        OnMouseDown: execute { SR_MulticarrierModule.udiSingleCarrierNr := 131; }
    Button (68,712 25x25), "132", colour toggle: SR_MulticarrierModule.aifVisFeedback[132].ifFeedbackConfiguration.xApplicationLoggerEntriesActive, invisible if: SR_MulticarrierModule.ifMulticarrier.ifFeedback.ifFeedbackConfiguration.udiNumberOfCarriers < 132
        toggle SR_MulticarrierModule.xSetSingleAplMsg
        OnMouseDown: execute { SR_MulticarrierModule.udiSingleCarrierNr := 132; }
    Button (108,712 25x25), "133", colour toggle: SR_MulticarrierModule.aifVisFeedback[133].ifFeedbackConfiguration.xApplicationLoggerEntriesActive, invisible if: SR_MulticarrierModule.ifMulticarrier.ifFeedback.ifFeedbackConfiguration.udiNumberOfCarriers < 133
        toggle SR_MulticarrierModule.xSetSingleAplMsg
        OnMouseDown: execute { SR_MulticarrierModule.udiSingleCarrierNr := 133; }
    Button (148,712 25x25), "134", colour toggle: SR_MulticarrierModule.aifVisFeedback[134].ifFeedbackConfiguration.xApplicationLoggerEntriesActive, invisible if: SR_MulticarrierModule.ifMulticarrier.ifFeedback.ifFeedbackConfiguration.udiNumberOfCarriers < 134
        toggle SR_MulticarrierModule.xSetSingleAplMsg
        OnMouseDown: execute { SR_MulticarrierModule.udiSingleCarrierNr := 134; }
    Button (188,712 25x25), "135", colour toggle: SR_MulticarrierModule.aifVisFeedback[135].ifFeedbackConfiguration.xApplicationLoggerEntriesActive, invisible if: SR_MulticarrierModule.ifMulticarrier.ifFeedback.ifFeedbackConfiguration.udiNumberOfCarriers < 135
        toggle SR_MulticarrierModule.xSetSingleAplMsg
        OnMouseDown: execute { SR_MulticarrierModule.udiSingleCarrierNr := 135; }
    Button (228,712 25x25), "136", colour toggle: SR_MulticarrierModule.aifVisFeedback[136].ifFeedbackConfiguration.xApplicationLoggerEntriesActive, invisible if: SR_MulticarrierModule.ifMulticarrier.ifFeedback.ifFeedbackConfiguration.udiNumberOfCarriers < 136
        toggle SR_MulticarrierModule.xSetSingleAplMsg
        OnMouseDown: execute { SR_MulticarrierModule.udiSingleCarrierNr := 136; }
    Button (268,712 25x25), "137", colour toggle: SR_MulticarrierModule.aifVisFeedback[137].ifFeedbackConfiguration.xApplicationLoggerEntriesActive, invisible if: SR_MulticarrierModule.ifMulticarrier.ifFeedback.ifFeedbackConfiguration.udiNumberOfCarriers < 137
        toggle SR_MulticarrierModule.xSetSingleAplMsg
        OnMouseDown: execute { SR_MulticarrierModule.udiSingleCarrierNr := 137; }
    Button (308,712 25x25), "138", colour toggle: SR_MulticarrierModule.aifVisFeedback[138].ifFeedbackConfiguration.xApplicationLoggerEntriesActive, invisible if: SR_MulticarrierModule.ifMulticarrier.ifFeedback.ifFeedbackConfiguration.udiNumberOfCarriers < 138
        toggle SR_MulticarrierModule.xSetSingleAplMsg
        OnMouseDown: execute { SR_MulticarrierModule.udiSingleCarrierNr := 138; }
    Button (348,712 25x25), "139", colour toggle: SR_MulticarrierModule.aifVisFeedback[139].ifFeedbackConfiguration.xApplicationLoggerEntriesActive, invisible if: SR_MulticarrierModule.ifMulticarrier.ifFeedback.ifFeedbackConfiguration.udiNumberOfCarriers < 139
        toggle SR_MulticarrierModule.xSetSingleAplMsg
        OnMouseDown: execute { SR_MulticarrierModule.udiSingleCarrierNr := 139; }
    Button (387,712 25x25), "140", colour toggle: SR_MulticarrierModule.aifVisFeedback[140].ifFeedbackConfiguration.xApplicationLoggerEntriesActive, invisible if: SR_MulticarrierModule.ifMulticarrier.ifFeedback.ifFeedbackConfiguration.udiNumberOfCarriers < 140
        toggle SR_MulticarrierModule.xSetSingleAplMsg
        OnMouseDown: execute { SR_MulticarrierModule.udiSingleCarrierNr := 140; }
    Button (27,752 25x25), "141", colour toggle: SR_MulticarrierModule.aifVisFeedback[141].ifFeedbackConfiguration.xApplicationLoggerEntriesActive, invisible if: SR_MulticarrierModule.ifMulticarrier.ifFeedback.ifFeedbackConfiguration.udiNumberOfCarriers < 141
        toggle SR_MulticarrierModule.xSetSingleAplMsg
        OnMouseDown: execute { SR_MulticarrierModule.udiSingleCarrierNr := 141; }
    Button (67,752 25x25), "142", colour toggle: SR_MulticarrierModule.aifVisFeedback[142].ifFeedbackConfiguration.xApplicationLoggerEntriesActive, invisible if: SR_MulticarrierModule.ifMulticarrier.ifFeedback.ifFeedbackConfiguration.udiNumberOfCarriers < 142
        toggle SR_MulticarrierModule.xSetSingleAplMsg
        OnMouseDown: execute { SR_MulticarrierModule.udiSingleCarrierNr := 142; }
    Button (107,752 25x25), "143", colour toggle: SR_MulticarrierModule.aifVisFeedback[143].ifFeedbackConfiguration.xApplicationLoggerEntriesActive, invisible if: SR_MulticarrierModule.ifMulticarrier.ifFeedback.ifFeedbackConfiguration.udiNumberOfCarriers < 143
        toggle SR_MulticarrierModule.xSetSingleAplMsg
        OnMouseDown: execute { SR_MulticarrierModule.udiSingleCarrierNr := 143; }
    Button (147,752 25x25), "144", colour toggle: SR_MulticarrierModule.aifVisFeedback[144].ifFeedbackConfiguration.xApplicationLoggerEntriesActive, invisible if: SR_MulticarrierModule.ifMulticarrier.ifFeedback.ifFeedbackConfiguration.udiNumberOfCarriers < 144
        toggle SR_MulticarrierModule.xSetSingleAplMsg
        OnMouseDown: execute { SR_MulticarrierModule.udiSingleCarrierNr := 144; }
    Button (187,752 25x25), "145", colour toggle: SR_MulticarrierModule.aifVisFeedback[145].ifFeedbackConfiguration.xApplicationLoggerEntriesActive, invisible if: SR_MulticarrierModule.ifMulticarrier.ifFeedback.ifFeedbackConfiguration.udiNumberOfCarriers < 145
        toggle SR_MulticarrierModule.xSetSingleAplMsg
        OnMouseDown: execute { SR_MulticarrierModule.udiSingleCarrierNr := 145; }
    Button (227,752 25x25), "146", colour toggle: SR_MulticarrierModule.aifVisFeedback[146].ifFeedbackConfiguration.xApplicationLoggerEntriesActive, invisible if: SR_MulticarrierModule.ifMulticarrier.ifFeedback.ifFeedbackConfiguration.udiNumberOfCarriers < 146
        toggle SR_MulticarrierModule.xSetSingleAplMsg
        OnMouseDown: execute { SR_MulticarrierModule.udiSingleCarrierNr := 146; }
    Button (267,752 25x25), "147", colour toggle: SR_MulticarrierModule.aifVisFeedback[147].ifFeedbackConfiguration.xApplicationLoggerEntriesActive, invisible if: SR_MulticarrierModule.ifMulticarrier.ifFeedback.ifFeedbackConfiguration.udiNumberOfCarriers < 147
        toggle SR_MulticarrierModule.xSetSingleAplMsg
        OnMouseDown: execute { SR_MulticarrierModule.udiSingleCarrierNr := 147; }
    Button (307,752 25x25), "148", colour toggle: SR_MulticarrierModule.aifVisFeedback[148].ifFeedbackConfiguration.xApplicationLoggerEntriesActive, invisible if: SR_MulticarrierModule.ifMulticarrier.ifFeedback.ifFeedbackConfiguration.udiNumberOfCarriers < 148
        toggle SR_MulticarrierModule.xSetSingleAplMsg
        OnMouseDown: execute { SR_MulticarrierModule.udiSingleCarrierNr := 148; }
    Button (347,752 25x25), "149", colour toggle: SR_MulticarrierModule.aifVisFeedback[149].ifFeedbackConfiguration.xApplicationLoggerEntriesActive, invisible if: SR_MulticarrierModule.ifMulticarrier.ifFeedback.ifFeedbackConfiguration.udiNumberOfCarriers < 149
        toggle SR_MulticarrierModule.xSetSingleAplMsg
        OnMouseDown: execute { SR_MulticarrierModule.udiSingleCarrierNr := 149; }
    Button (388,752 25x25), "150", colour toggle: SR_MulticarrierModule.aifVisFeedback[150].ifFeedbackConfiguration.xApplicationLoggerEntriesActive, invisible if: SR_MulticarrierModule.ifMulticarrier.ifFeedback.ifFeedbackConfiguration.udiNumberOfCarriers < 150
        toggle SR_MulticarrierModule.xSetSingleAplMsg
        OnMouseDown: execute { SR_MulticarrierModule.udiSingleCarrierNr := 150; }
    Button (188,672 25x25), "125", colour toggle: SR_MulticarrierModule.aifVisFeedback[125].ifFeedbackConfiguration.xApplicationLoggerEntriesActive, invisible if: SR_MulticarrierModule.ifMulticarrier.ifFeedback.ifFeedbackConfiguration.udiNumberOfCarriers < 125
        toggle SR_MulticarrierModule.xSetSingleAplMsg
        OnMouseDown: execute { SR_MulticarrierModule.udiSingleCarrierNr := 125; }
    Button (228,672 25x25), "126", colour toggle: SR_MulticarrierModule.aifVisFeedback[126].ifFeedbackConfiguration.xApplicationLoggerEntriesActive, invisible if: SR_MulticarrierModule.ifMulticarrier.ifFeedback.ifFeedbackConfiguration.udiNumberOfCarriers < 126
        toggle SR_MulticarrierModule.xSetSingleAplMsg
        OnMouseDown: execute { SR_MulticarrierModule.udiSingleCarrierNr := 126; }
    Button (268,672 25x25), "127", colour toggle: SR_MulticarrierModule.aifVisFeedback[127].ifFeedbackConfiguration.xApplicationLoggerEntriesActive, invisible if: SR_MulticarrierModule.ifMulticarrier.ifFeedback.ifFeedbackConfiguration.udiNumberOfCarriers < 127
        toggle SR_MulticarrierModule.xSetSingleAplMsg
        OnMouseDown: execute { SR_MulticarrierModule.udiSingleCarrierNr := 127; }
    Button (308,672 25x25), "128", colour toggle: SR_MulticarrierModule.aifVisFeedback[128].ifFeedbackConfiguration.xApplicationLoggerEntriesActive, invisible if: SR_MulticarrierModule.ifMulticarrier.ifFeedback.ifFeedbackConfiguration.udiNumberOfCarriers < 128
        toggle SR_MulticarrierModule.xSetSingleAplMsg
        OnMouseDown: execute { SR_MulticarrierModule.udiSingleCarrierNr := 128; }
    Button (348,672 25x25), "129", colour toggle: SR_MulticarrierModule.aifVisFeedback[129].ifFeedbackConfiguration.xApplicationLoggerEntriesActive, invisible if: SR_MulticarrierModule.ifMulticarrier.ifFeedback.ifFeedbackConfiguration.udiNumberOfCarriers < 129
        toggle SR_MulticarrierModule.xSetSingleAplMsg
        OnMouseDown: execute { SR_MulticarrierModule.udiSingleCarrierNr := 129; }
    Rectangle (339,110 100x20), "End: %0.0f", text variable: SR_MulticarrierModule.lrAplEndTrackPos
        OnMouseClick: write the text variable via Default, min 0, max SR_MulticarrierModule.fbMulticarrier.ifFeedback.ifFeedbackConfiguration.lrTrackLength
    Button (339,49 100x40), "Set entries by Position", colour toggle: SR_MultiCarriermodule.xAplMsgStartPosAndEndPos
        toggle SR_MultiCarriermodule.xAplMsgStartPosAndEndPos
    Rectangle (339,90 100x20), "Start: %0.0f", text variable: SR_MulticarrierModule.lrAplStartTrackPos
        OnMouseClick: write the text variable via Default, min 0, max SR_MulticarrierModule.fbMulticarrier.ifFeedback.ifFeedbackConfiguration.lrTrackLength
END_VISUALIZATION

// LMC_PacDrive/Application/TemplateFullProgrammingFramework/Visualization/Multicarrier/Vis_Error
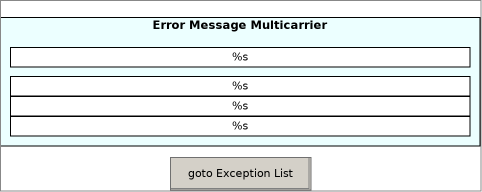
VISUALIZATION Vis_Error  // 482x192
    Rectangle (0,17 480x129), "Error Message Multicarrier"
    Rectangle (10,47 460x20), "%s", text variable: SR_MultiCarrierModule.stException.sDiagExt
    Rectangle (10,76 460x20), "%s", text variable: SR_MultiCarrierModule.sResultMsg1
    Rectangle (10,96 460x20), "%s", text variable: SR_MultiCarrierModule.sResultMsg2
    Button (170,157 141x33), "goto Exception List"
        OnMouseClick:  Assign=VIS_ExceptionList, Type=Assignment
    Rectangle (10,116 460x20), "%s", text variable: SR_MultiCarrierModule.sResultMsg3
END_VISUALIZATION

// LMC_PacDrive/Application/TemplateFullProgrammingFramework/Visualization/Multicarrier/Vis_Jogging
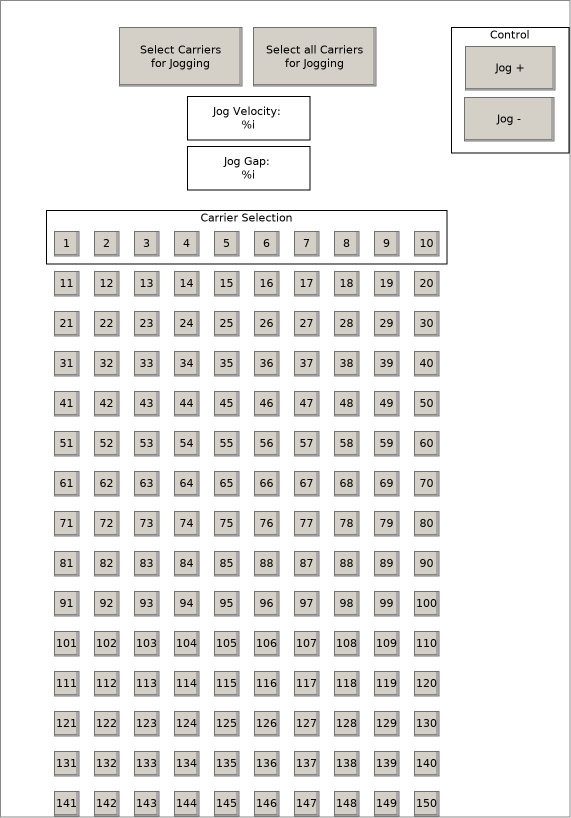
VISUALIZATION Vis_Jogging  // 571x818
    Rectangle (451,27 118x126), "Control", input disabled if: NOT SR_MainMachine.xActManual
    Button (465,46 90x44), "Jog +", colour toggle: SR_MulticarrierModule.xJogForw, input disabled if: NOT SR_MainMachine.xActManual
        tap SR_MulticarrierModule.xJogForw
    Button (464,97 90x44), "Jog -", colour toggle: SR_MulticarrierModule.xJogBack, input disabled if: NOT SR_MainMachine.xActManual
        tap SR_MulticarrierModule.xJogBack p3779583253=TRUE
    Button (119,27 123x59), "Select Carriers for Jogging", colour toggle: SR_MulticarrierModule.xJogSingleCarrier, input disabled if: NOT SR_MainMachine.xActManual
        tap SR_MultiCarriermodule.xSetJogSingleCarrier
    Button (253,27 123x59), "Select all Carriers for Jogging", colour toggle: SR_MulticarrierModule.xJogAllCarrier, input disabled if: NOT SR_MainMachine.xActManual
        tap SR_MulticarrierModule.xSetJogAllCarrier
    Rectangle (187,96 123x44), "Jog Velocity: %i", tooltip "Acc = Velocity Dec = Velocity x 10 Jerk = Velocity x 100", text variable: SR_MulticarrierModule.lrJogVelocity, input disabled if: NOT SR_MainMachine.xActManual
        OnMouseClick: write the text variable via Default, min 0
    Rectangle (187,146 123x44), "Jog Gap: %i", tooltip "Jog possible when Actual Gap >= Jog Gap (Decelerate moving Carrier when Actual Gap < Jog Gap)", text variable: SR_MulticarrierModule.lrJogMinDistanceBetweenCarrier, invisible if: SR_MulticarrierModule.xJogAllCarrier, input disabled if: NOT SR_MainMachine.xActManual
        OnMouseClick: write the text variable via Default, min 0
    Rectangle (46,210 401x54), "Carrier Selection"
        p1126004900: SR_MultiCarriermodule.udiDeltaBottomY
    Button (54,231 25x25), "1", colour toggle: SR_MultiCarrierModule.aifVisFeedback[1].ifFeedbackJogging.xJogActivated, invisible if: SR_MulticarrierModule.ifMulticarrier.ifFeedback.ifFeedbackConfiguration.udiNumberOfCarriers < 1, input disabled if: NOT SR_MainMachine.xActManual
        toggle SR_MultiCarriermodule.xSetCarrierForJoggingFromVis
        OnMouseClick: execute { SR_MultiCarrierModule.udiJoggingCarrierNr := 1; }
    Button (94,231 25x25), "2", colour toggle: SR_MultiCarrierModule.aifVisFeedback[2].ifFeedbackJogging.xJogActivated, invisible if: SR_MulticarrierModule.ifMulticarrier.ifFeedback.ifFeedbackConfiguration.udiNumberOfCarriers < 2, input disabled if: NOT SR_MainMachine.xActManual
        toggle SR_MultiCarriermodule.xSetCarrierForJoggingFromVis
        OnMouseClick: execute { SR_MultiCarrierModule.udiJoggingCarrierNr := 2; }
    Button (134,231 25x25), "3", colour toggle: SR_MultiCarrierModule.aifVisFeedback[3].ifFeedbackJogging.xJogActivated, invisible if: SR_MulticarrierModule.ifMulticarrier.ifFeedback.ifFeedbackConfiguration.udiNumberOfCarriers < 3, input disabled if: NOT SR_MainMachine.xActManual
        toggle SR_MultiCarriermodule.xSetCarrierForJoggingFromVis
        OnMouseClick: execute { SR_MultiCarrierModule.udiJoggingCarrierNr := 3; }
    Button (174,231 25x25), "4", colour toggle: SR_MultiCarrierModule.aifVisFeedback[4].ifFeedbackJogging.xJogActivated, invisible if: SR_MulticarrierModule.ifMulticarrier.ifFeedback.ifFeedbackConfiguration.udiNumberOfCarriers < 4, input disabled if: NOT SR_MainMachine.xActManual
        toggle SR_MultiCarriermodule.xSetCarrierForJoggingFromVis
        OnMouseClick: execute { SR_MultiCarrierModule.udiJoggingCarrierNr := 4; }
    Button (214,231 25x25), "5", colour toggle: SR_MultiCarrierModule.aifVisFeedback[5].ifFeedbackJogging.xJogActivated, invisible if: SR_MulticarrierModule.ifMulticarrier.ifFeedback.ifFeedbackConfiguration.udiNumberOfCarriers < 5, input disabled if: NOT SR_MainMachine.xActManual
        toggle SR_MultiCarriermodule.xSetCarrierForJoggingFromVis
        OnMouseClick: execute { SR_MultiCarrierModule.udiJoggingCarrierNr := 5; }
    Button (254,231 25x25), "6", colour toggle: SR_MultiCarrierModule.aifVisFeedback[6].ifFeedbackJogging.xJogActivated, invisible if: SR_MulticarrierModule.ifMulticarrier.ifFeedback.ifFeedbackConfiguration.udiNumberOfCarriers < 6, input disabled if: NOT SR_MainMachine.xActManual
        toggle SR_MultiCarriermodule.xSetCarrierForJoggingFromVis
        OnMouseClick: execute { SR_MultiCarrierModule.udiJoggingCarrierNr := 6; }
    Button (294,231 25x25), "7", colour toggle: SR_MultiCarrierModule.aifVisFeedback[7].ifFeedbackJogging.xJogActivated, invisible if: SR_MulticarrierModule.ifMulticarrier.ifFeedback.ifFeedbackConfiguration.udiNumberOfCarriers < 7, input disabled if: NOT SR_MainMachine.xActManual
        toggle SR_MultiCarriermodule.xSetCarrierForJoggingFromVis
        OnMouseClick: execute { SR_MultiCarrierModule.udiJoggingCarrierNr := 7; }
    Button (334,231 25x25), "8", colour toggle: SR_MultiCarrierModule.aifVisFeedback[8].ifFeedbackJogging.xJogActivated, invisible if: SR_MulticarrierModule.ifMulticarrier.ifFeedback.ifFeedbackConfiguration.udiNumberOfCarriers < 8, input disabled if: NOT SR_MainMachine.xActManual
        toggle SR_MultiCarriermodule.xSetCarrierForJoggingFromVis
        OnMouseClick: execute { SR_MultiCarrierModule.udiJoggingCarrierNr := 8; }
    Button (374,231 25x25), "9", colour toggle: SR_MultiCarrierModule.aifVisFeedback[9].ifFeedbackJogging.xJogActivated, invisible if: SR_MulticarrierModule.ifMulticarrier.ifFeedback.ifFeedbackConfiguration.udiNumberOfCarriers < 9, input disabled if: NOT SR_MainMachine.xActManual
        toggle SR_MultiCarriermodule.xSetCarrierForJoggingFromVis
        OnMouseClick: execute { SR_MultiCarrierModule.udiJoggingCarrierNr := 9; }
    Button (414,231 25x25), "10", colour toggle: SR_MultiCarrierModule.aifVisFeedback[10].ifFeedbackJogging.xJogActivated, invisible if: SR_MulticarrierModule.ifMulticarrier.ifFeedback.ifFeedbackConfiguration.udiNumberOfCarriers < 10, input disabled if: NOT SR_MainMachine.xActManual
        toggle SR_MultiCarriermodule.xSetCarrierForJoggingFromVis
        OnMouseClick: execute { SR_MultiCarrierModule.udiJoggingCarrierNr := 10; }
    Button (414,271 25x25), "20", colour toggle: SR_MultiCarrierModule.aifVisFeedback[20].ifFeedbackJogging.xJogActivated, invisible if: SR_MulticarrierModule.ifMulticarrier.ifFeedback.ifFeedbackConfiguration.udiNumberOfCarriers < 20, input disabled if: NOT SR_MainMachine.xActManual
        toggle SR_MultiCarriermodule.xSetCarrierForJoggingFromVis
        OnMouseClick: execute { SR_MultiCarrierModule.udiJoggingCarrierNr := 20; }
    Button (414,311 25x25), "30", colour toggle: SR_MultiCarrierModule.aifVisFeedback[30].ifFeedbackJogging.xJogActivated, invisible if: SR_MulticarrierModule.ifMulticarrier.ifFeedback.ifFeedbackConfiguration.udiNumberOfCarriers < 30, input disabled if: NOT SR_MainMachine.xActManual
        toggle SR_MultiCarriermodule.xSetCarrierForJoggingFromVis
        OnMouseClick: execute { SR_MultiCarrierModule.udiJoggingCarrierNr := 30; }
    Button (414,351 25x25), "40", colour toggle: SR_MultiCarrierModule.aifVisFeedback[40].ifFeedbackJogging.xJogActivated, invisible if: SR_MulticarrierModule.ifMulticarrier.ifFeedback.ifFeedbackConfiguration.udiNumberOfCarriers < 40, input disabled if: NOT SR_MainMachine.xActManual
        toggle SR_MultiCarriermodule.xSetCarrierForJoggingFromVis
        OnMouseClick: execute { SR_MultiCarrierModule.udiJoggingCarrierNr := 40; }
    Button (414,391 25x25), "50", colour toggle: SR_MultiCarrierModule.aifVisFeedback[50].ifFeedbackJogging.xJogActivated, invisible if: SR_MulticarrierModule.ifMulticarrier.ifFeedback.ifFeedbackConfiguration.udiNumberOfCarriers < 50, input disabled if: NOT SR_MainMachine.xActManual
        toggle SR_MultiCarriermodule.xSetCarrierForJoggingFromVis
        OnMouseClick: execute { SR_MultiCarrierModule.udiJoggingCarrierNr := 50; }
    Button (414,431 25x25), "60", colour toggle: SR_MultiCarrierModule.aifVisFeedback[60].ifFeedbackJogging.xJogActivated, invisible if: SR_MulticarrierModule.ifMulticarrier.ifFeedback.ifFeedbackConfiguration.udiNumberOfCarriers < 60, input disabled if: NOT SR_MainMachine.xActManual
        toggle SR_MultiCarriermodule.xSetCarrierForJoggingFromVis
        OnMouseClick: execute { SR_MultiCarrierModule.udiJoggingCarrierNr := 60; }
    Button (54,471 25x25), "61", colour toggle: SR_MultiCarrierModule.aifVisFeedback[61].ifFeedbackJogging.xJogActivated, invisible if: SR_MulticarrierModule.ifMulticarrier.ifFeedback.ifFeedbackConfiguration.udiNumberOfCarriers < 61, input disabled if: NOT SR_MainMachine.xActManual
        toggle SR_MultiCarriermodule.xSetCarrierForJoggingFromVis
        OnMouseClick: execute { SR_MultiCarrierModule.udiJoggingCarrierNr := 61; }
    Button (94,471 25x25), "62", colour toggle: SR_MultiCarrierModule.aifVisFeedback[62].ifFeedbackJogging.xJogActivated, invisible if: SR_MulticarrierModule.ifMulticarrier.ifFeedback.ifFeedbackConfiguration.udiNumberOfCarriers < 62, input disabled if: NOT SR_MainMachine.xActManual
        toggle SR_MultiCarriermodule.xSetCarrierForJoggingFromVis
        OnMouseClick: execute { SR_MultiCarrierModule.udiJoggingCarrierNr := 62; }
    Button (134,471 25x25), "63", colour toggle: SR_MultiCarrierModule.aifVisFeedback[63].ifFeedbackJogging.xJogActivated, invisible if: SR_MulticarrierModule.ifMulticarrier.ifFeedback.ifFeedbackConfiguration.udiNumberOfCarriers < 63, input disabled if: NOT SR_MainMachine.xActManual
        toggle SR_MultiCarriermodule.xSetCarrierForJoggingFromVis
        OnMouseClick: execute { SR_MultiCarrierModule.udiJoggingCarrierNr := 63; }
    Button (174,471 25x25), "64", colour toggle: SR_MultiCarrierModule.aifVisFeedback[64].ifFeedbackJogging.xJogActivated, invisible if: SR_MulticarrierModule.ifMulticarrier.ifFeedback.ifFeedbackConfiguration.udiNumberOfCarriers < 64, input disabled if: NOT SR_MainMachine.xActManual
        toggle SR_MultiCarriermodule.xSetCarrierForJoggingFromVis
        OnMouseClick: execute { SR_MultiCarrierModule.udiJoggingCarrierNr := 64; }
    Button (214,471 25x25), "65", colour toggle: SR_MultiCarrierModule.aifVisFeedback[65].ifFeedbackJogging.xJogActivated, invisible if: SR_MulticarrierModule.ifMulticarrier.ifFeedback.ifFeedbackConfiguration.udiNumberOfCarriers < 65, input disabled if: NOT SR_MainMachine.xActManual
        toggle SR_MultiCarriermodule.xSetCarrierForJoggingFromVis
        OnMouseClick: execute { SR_MultiCarrierModule.udiJoggingCarrierNr := 65; }
    Button (254,471 25x25), "66", colour toggle: SR_MultiCarrierModule.aifVisFeedback[66].ifFeedbackJogging.xJogActivated, invisible if: SR_MulticarrierModule.ifMulticarrier.ifFeedback.ifFeedbackConfiguration.udiNumberOfCarriers < 66, input disabled if: NOT SR_MainMachine.xActManual
        toggle SR_MultiCarriermodule.xSetCarrierForJoggingFromVis
        OnMouseClick: execute { SR_MultiCarrierModule.udiJoggingCarrierNr := 66; }
    Button (294,471 25x25), "67", colour toggle: SR_MultiCarrierModule.aifVisFeedback[67].ifFeedbackJogging.xJogActivated, invisible if: SR_MulticarrierModule.ifMulticarrier.ifFeedback.ifFeedbackConfiguration.udiNumberOfCarriers < 67, input disabled if: NOT SR_MainMachine.xActManual
        toggle SR_MultiCarriermodule.xSetCarrierForJoggingFromVis
        OnMouseClick: execute { SR_MultiCarrierModule.udiJoggingCarrierNr := 67; }
    Button (334,471 25x25), "68", colour toggle: SR_MultiCarrierModule.aifVisFeedback[68].ifFeedbackJogging.xJogActivated, invisible if: SR_MulticarrierModule.ifMulticarrier.ifFeedback.ifFeedbackConfiguration.udiNumberOfCarriers < 68, input disabled if: NOT SR_MainMachine.xActManual
        toggle SR_MultiCarriermodule.xSetCarrierForJoggingFromVis
        OnMouseClick: execute { SR_MultiCarrierModule.udiJoggingCarrierNr := 68; }
    Button (374,471 25x25), "69", colour toggle: SR_MultiCarrierModule.aifVisFeedback[69].ifFeedbackJogging.xJogActivated, invisible if: SR_MulticarrierModule.ifMulticarrier.ifFeedback.ifFeedbackConfiguration.udiNumberOfCarriers < 69, input disabled if: NOT SR_MainMachine.xActManual
        toggle SR_MultiCarriermodule.xSetCarrierForJoggingFromVis
        OnMouseClick: execute { SR_MultiCarrierModule.udiJoggingCarrierNr := 69; }
    Button (414,471 25x25), "70", colour toggle: SR_MultiCarrierModule.aifVisFeedback[70].ifFeedbackJogging.xJogActivated, invisible if: SR_MulticarrierModule.ifMulticarrier.ifFeedback.ifFeedbackConfiguration.udiNumberOfCarriers < 70, input disabled if: NOT SR_MainMachine.xActManual
        toggle SR_MultiCarriermodule.xSetCarrierForJoggingFromVis
        OnMouseClick: execute { SR_MultiCarrierModule.udiJoggingCarrierNr := 70; }
    Button (54,271 25x25), "11", colour toggle: SR_MultiCarrierModule.aifVisFeedback[11].ifFeedbackJogging.xJogActivated, invisible if: SR_MulticarrierModule.ifMulticarrier.ifFeedback.ifFeedbackConfiguration.udiNumberOfCarriers < 11, input disabled if: NOT SR_MainMachine.xActManual
        toggle SR_MultiCarriermodule.xSetCarrierForJoggingFromVis
        OnMouseClick: execute { SR_MultiCarrierModule.udiJoggingCarrierNr := 11; }
    Button (94,271 25x25), "12", colour toggle: SR_MultiCarrierModule.aifVisFeedback[12].ifFeedbackJogging.xJogActivated, invisible if: SR_MulticarrierModule.ifMulticarrier.ifFeedback.ifFeedbackConfiguration.udiNumberOfCarriers < 12, input disabled if: NOT SR_MainMachine.xActManual
        toggle SR_MultiCarriermodule.xSetCarrierForJoggingFromVis
        OnMouseClick: execute { SR_MultiCarrierModule.udiJoggingCarrierNr := 12; }
    Button (134,271 25x25), "13", colour toggle: SR_MultiCarrierModule.aifVisFeedback[13].ifFeedbackJogging.xJogActivated, invisible if: SR_MulticarrierModule.ifMulticarrier.ifFeedback.ifFeedbackConfiguration.udiNumberOfCarriers < 13, input disabled if: NOT SR_MainMachine.xActManual
        toggle SR_MultiCarriermodule.xSetCarrierForJoggingFromVis
        OnMouseClick: execute { SR_MultiCarrierModule.udiJoggingCarrierNr := 13; }
    Button (174,271 25x25), "14", colour toggle: SR_MultiCarrierModule.aifVisFeedback[14].ifFeedbackJogging.xJogActivated, invisible if: SR_MulticarrierModule.ifMulticarrier.ifFeedback.ifFeedbackConfiguration.udiNumberOfCarriers < 14, input disabled if: NOT SR_MainMachine.xActManual
        toggle SR_MultiCarriermodule.xSetCarrierForJoggingFromVis
        OnMouseClick: execute { SR_MultiCarrierModule.udiJoggingCarrierNr := 14; }
    Button (214,271 25x25), "15", colour toggle: SR_MultiCarrierModule.aifVisFeedback[15].ifFeedbackJogging.xJogActivated, invisible if: SR_MulticarrierModule.ifMulticarrier.ifFeedback.ifFeedbackConfiguration.udiNumberOfCarriers < 15, input disabled if: NOT SR_MainMachine.xActManual
        toggle SR_MultiCarriermodule.xSetCarrierForJoggingFromVis
        OnMouseClick: execute { SR_MultiCarrierModule.udiJoggingCarrierNr := 15; }
    Button (254,271 25x25), "16", colour toggle: SR_MultiCarrierModule.aifVisFeedback[16].ifFeedbackJogging.xJogActivated, invisible if: SR_MulticarrierModule.ifMulticarrier.ifFeedback.ifFeedbackConfiguration.udiNumberOfCarriers < 16, input disabled if: NOT SR_MainMachine.xActManual
        toggle SR_MultiCarriermodule.xSetCarrierForJoggingFromVis
        OnMouseClick: execute { SR_MultiCarrierModule.udiJoggingCarrierNr := 16; }
    Button (294,271 25x25), "17", colour toggle: SR_MultiCarrierModule.aifVisFeedback[17].ifFeedbackJogging.xJogActivated, invisible if: SR_MulticarrierModule.ifMulticarrier.ifFeedback.ifFeedbackConfiguration.udiNumberOfCarriers < 17, input disabled if: NOT SR_MainMachine.xActManual
        toggle SR_MultiCarriermodule.xSetCarrierForJoggingFromVis
        OnMouseClick: execute { SR_MultiCarrierModule.udiJoggingCarrierNr := 17; }
    Button (334,271 25x25), "18", colour toggle: SR_MultiCarrierModule.aifVisFeedback[18].ifFeedbackJogging.xJogActivated, invisible if: SR_MulticarrierModule.ifMulticarrier.ifFeedback.ifFeedbackConfiguration.udiNumberOfCarriers < 18, input disabled if: NOT SR_MainMachine.xActManual
        toggle SR_MultiCarriermodule.xSetCarrierForJoggingFromVis
        OnMouseClick: execute { SR_MultiCarrierModule.udiJoggingCarrierNr := 18; }
    Button (374,271 25x25), "19", colour toggle: SR_MultiCarrierModule.aifVisFeedback[19].ifFeedbackJogging.xJogActivated, invisible if: SR_MulticarrierModule.ifMulticarrier.ifFeedback.ifFeedbackConfiguration.udiNumberOfCarriers < 19, input disabled if: NOT SR_MainMachine.xActManual
        toggle SR_MultiCarriermodule.xSetCarrierForJoggingFromVis
        OnMouseClick: execute { SR_MultiCarrierModule.udiJoggingCarrierNr := 19; }
    Button (54,311 25x25), "21", colour toggle: SR_MultiCarrierModule.aifVisFeedback[21].ifFeedbackJogging.xJogActivated, invisible if: SR_MulticarrierModule.ifMulticarrier.ifFeedback.ifFeedbackConfiguration.udiNumberOfCarriers < 21, input disabled if: NOT SR_MainMachine.xActManual
        toggle SR_MultiCarriermodule.xSetCarrierForJoggingFromVis
        OnMouseClick: execute { SR_MultiCarrierModule.udiJoggingCarrierNr := 21; }
    Button (94,311 25x25), "22", colour toggle: SR_MultiCarrierModule.aifVisFeedback[22].ifFeedbackJogging.xJogActivated, invisible if: SR_MulticarrierModule.ifMulticarrier.ifFeedback.ifFeedbackConfiguration.udiNumberOfCarriers < 22, input disabled if: NOT SR_MainMachine.xActManual
        toggle SR_MultiCarriermodule.xSetCarrierForJoggingFromVis
        OnMouseClick: execute { SR_MultiCarrierModule.udiJoggingCarrierNr := 22; }
    Button (134,311 25x25), "23", colour toggle: SR_MultiCarrierModule.aifVisFeedback[23].ifFeedbackJogging.xJogActivated, invisible if: SR_MulticarrierModule.ifMulticarrier.ifFeedback.ifFeedbackConfiguration.udiNumberOfCarriers < 23, input disabled if: NOT SR_MainMachine.xActManual
        toggle SR_MultiCarriermodule.xSetCarrierForJoggingFromVis
        OnMouseClick: execute { SR_MultiCarrierModule.udiJoggingCarrierNr := 23; }
    Button (174,311 25x25), "24", colour toggle: SR_MultiCarrierModule.aifVisFeedback[24].ifFeedbackJogging.xJogActivated, invisible if: SR_MulticarrierModule.ifMulticarrier.ifFeedback.ifFeedbackConfiguration.udiNumberOfCarriers < 24, input disabled if: NOT SR_MainMachine.xActManual
        toggle SR_MultiCarriermodule.xSetCarrierForJoggingFromVis
        OnMouseClick: execute { SR_MultiCarrierModule.udiJoggingCarrierNr := 24; }
    Button (214,311 25x25), "25", colour toggle: SR_MultiCarrierModule.aifVisFeedback[25].ifFeedbackJogging.xJogActivated, invisible if: SR_MulticarrierModule.ifMulticarrier.ifFeedback.ifFeedbackConfiguration.udiNumberOfCarriers < 25, input disabled if: NOT SR_MainMachine.xActManual
        toggle SR_MultiCarriermodule.xSetCarrierForJoggingFromVis
        OnMouseClick: execute { SR_MultiCarrierModule.udiJoggingCarrierNr := 25; }
    Button (254,311 25x25), "26", colour toggle: SR_MultiCarrierModule.aifVisFeedback[26].ifFeedbackJogging.xJogActivated, invisible if: SR_MulticarrierModule.ifMulticarrier.ifFeedback.ifFeedbackConfiguration.udiNumberOfCarriers < 26, input disabled if: NOT SR_MainMachine.xActManual
        toggle SR_MultiCarriermodule.xSetCarrierForJoggingFromVis
        OnMouseClick: execute { SR_MultiCarrierModule.udiJoggingCarrierNr := 26; }
    Button (294,311 25x25), "27", colour toggle: SR_MultiCarrierModule.aifVisFeedback[27].ifFeedbackJogging.xJogActivated, invisible if: SR_MulticarrierModule.ifMulticarrier.ifFeedback.ifFeedbackConfiguration.udiNumberOfCarriers < 27, input disabled if: NOT SR_MainMachine.xActManual
        toggle SR_MultiCarriermodule.xSetCarrierForJoggingFromVis
        OnMouseClick: execute { SR_MultiCarrierModule.udiJoggingCarrierNr := 27; }
    Button (334,311 25x25), "28", colour toggle: SR_MultiCarrierModule.aifVisFeedback[28].ifFeedbackJogging.xJogActivated, invisible if: SR_MulticarrierModule.ifMulticarrier.ifFeedback.ifFeedbackConfiguration.udiNumberOfCarriers < 28, input disabled if: NOT SR_MainMachine.xActManual
        toggle SR_MultiCarriermodule.xSetCarrierForJoggingFromVis
        OnMouseClick: execute { SR_MultiCarrierModule.udiJoggingCarrierNr := 28; }
    Button (374,311 25x25), "29", colour toggle: SR_MultiCarrierModule.aifVisFeedback[29].ifFeedbackJogging.xJogActivated, invisible if: SR_MulticarrierModule.ifMulticarrier.ifFeedback.ifFeedbackConfiguration.udiNumberOfCarriers < 29, input disabled if: NOT SR_MainMachine.xActManual
        toggle SR_MultiCarriermodule.xSetCarrierForJoggingFromVis
        OnMouseClick: execute { SR_MultiCarrierModule.udiJoggingCarrierNr := 29; }
    Button (54,351 25x25), "31", colour toggle: SR_MultiCarrierModule.aifVisFeedback[31].ifFeedbackJogging.xJogActivated, invisible if: SR_MulticarrierModule.ifMulticarrier.ifFeedback.ifFeedbackConfiguration.udiNumberOfCarriers < 31, input disabled if: NOT SR_MainMachine.xActManual
        toggle SR_MultiCarriermodule.xSetCarrierForJoggingFromVis
        OnMouseClick: execute { SR_MultiCarrierModule.udiJoggingCarrierNr := 31; }
    Button (94,351 25x25), "32", colour toggle: SR_MultiCarrierModule.aifVisFeedback[32].ifFeedbackJogging.xJogActivated, invisible if: SR_MulticarrierModule.ifMulticarrier.ifFeedback.ifFeedbackConfiguration.udiNumberOfCarriers < 32, input disabled if: NOT SR_MainMachine.xActManual
        toggle SR_MultiCarriermodule.xSetCarrierForJoggingFromVis
        OnMouseClick: execute { SR_MultiCarrierModule.udiJoggingCarrierNr := 32; }
    Button (134,351 25x25), "33", colour toggle: SR_MultiCarrierModule.aifVisFeedback[33].ifFeedbackJogging.xJogActivated, invisible if: SR_MulticarrierModule.ifMulticarrier.ifFeedback.ifFeedbackConfiguration.udiNumberOfCarriers < 33, input disabled if: NOT SR_MainMachine.xActManual
        toggle SR_MultiCarriermodule.xSetCarrierForJoggingFromVis
        OnMouseClick: execute { SR_MultiCarrierModule.udiJoggingCarrierNr := 33; }
    Button (174,351 25x25), "34", colour toggle: SR_MultiCarrierModule.aifVisFeedback[34].ifFeedbackJogging.xJogActivated, invisible if: SR_MulticarrierModule.ifMulticarrier.ifFeedback.ifFeedbackConfiguration.udiNumberOfCarriers < 34, input disabled if: NOT SR_MainMachine.xActManual
        toggle SR_MultiCarriermodule.xSetCarrierForJoggingFromVis
        OnMouseClick: execute { SR_MultiCarrierModule.udiJoggingCarrierNr := 34; }
    Button (214,351 25x25), "35", colour toggle: SR_MultiCarrierModule.aifVisFeedback[35].ifFeedbackJogging.xJogActivated, invisible if: SR_MulticarrierModule.ifMulticarrier.ifFeedback.ifFeedbackConfiguration.udiNumberOfCarriers < 35, input disabled if: NOT SR_MainMachine.xActManual
        toggle SR_MultiCarriermodule.xSetCarrierForJoggingFromVis
        OnMouseClick: execute { SR_MultiCarrierModule.udiJoggingCarrierNr := 35; }
    Button (254,351 25x25), "36", colour toggle: SR_MultiCarrierModule.aifVisFeedback[36].ifFeedbackJogging.xJogActivated, invisible if: SR_MulticarrierModule.ifMulticarrier.ifFeedback.ifFeedbackConfiguration.udiNumberOfCarriers < 36, input disabled if: NOT SR_MainMachine.xActManual
        toggle SR_MultiCarriermodule.xSetCarrierForJoggingFromVis
        OnMouseClick: execute { SR_MultiCarrierModule.udiJoggingCarrierNr := 36; }
    Button (294,351 25x25), "37", colour toggle: SR_MultiCarrierModule.aifVisFeedback[37].ifFeedbackJogging.xJogActivated, invisible if: SR_MulticarrierModule.ifMulticarrier.ifFeedback.ifFeedbackConfiguration.udiNumberOfCarriers < 37, input disabled if: NOT SR_MainMachine.xActManual
        toggle SR_MultiCarriermodule.xSetCarrierForJoggingFromVis
        OnMouseClick: execute { SR_MultiCarrierModule.udiJoggingCarrierNr := 37; }
    Button (334,351 25x25), "38", colour toggle: SR_MultiCarrierModule.aifVisFeedback[38].ifFeedbackJogging.xJogActivated, invisible if: SR_MulticarrierModule.ifMulticarrier.ifFeedback.ifFeedbackConfiguration.udiNumberOfCarriers < 38, input disabled if: NOT SR_MainMachine.xActManual
        toggle SR_MultiCarriermodule.xSetCarrierForJoggingFromVis
        OnMouseClick: execute { SR_MultiCarrierModule.udiJoggingCarrierNr := 38; }
    Button (374,351 25x25), "39", colour toggle: SR_MultiCarrierModule.aifVisFeedback[39].ifFeedbackJogging.xJogActivated, invisible if: SR_MulticarrierModule.ifMulticarrier.ifFeedback.ifFeedbackConfiguration.udiNumberOfCarriers < 39, input disabled if: NOT SR_MainMachine.xActManual
        toggle SR_MultiCarriermodule.xSetCarrierForJoggingFromVis
        OnMouseClick: execute { SR_MultiCarrierModule.udiJoggingCarrierNr := 39; }
    Button (54,391 25x25), "41", colour toggle: SR_MultiCarrierModule.aifVisFeedback[41].ifFeedbackJogging.xJogActivated, invisible if: SR_MulticarrierModule.ifMulticarrier.ifFeedback.ifFeedbackConfiguration.udiNumberOfCarriers < 41, input disabled if: NOT SR_MainMachine.xActManual
        toggle SR_MultiCarriermodule.xSetCarrierForJoggingFromVis
        OnMouseClick: execute { SR_MultiCarrierModule.udiJoggingCarrierNr := 41; }
    Button (94,391 25x25), "42", colour toggle: SR_MultiCarrierModule.aifVisFeedback[42].ifFeedbackJogging.xJogActivated, invisible if: SR_MulticarrierModule.ifMulticarrier.ifFeedback.ifFeedbackConfiguration.udiNumberOfCarriers < 42, input disabled if: NOT SR_MainMachine.xActManual
        toggle SR_MultiCarriermodule.xSetCarrierForJoggingFromVis
        OnMouseClick: execute { SR_MultiCarrierModule.udiJoggingCarrierNr := 42; }
    Button (134,391 25x25), "43", colour toggle: SR_MultiCarrierModule.aifVisFeedback[43].ifFeedbackJogging.xJogActivated, invisible if: SR_MulticarrierModule.ifMulticarrier.ifFeedback.ifFeedbackConfiguration.udiNumberOfCarriers < 43, input disabled if: NOT SR_MainMachine.xActManual
        toggle SR_MultiCarriermodule.xSetCarrierForJoggingFromVis
        OnMouseClick: execute { SR_MultiCarrierModule.udiJoggingCarrierNr := 43; }
    Button (174,391 25x25), "44", colour toggle: SR_MultiCarrierModule.aifVisFeedback[44].ifFeedbackJogging.xJogActivated, invisible if: SR_MulticarrierModule.ifMulticarrier.ifFeedback.ifFeedbackConfiguration.udiNumberOfCarriers < 44, input disabled if: NOT SR_MainMachine.xActManual
        toggle SR_MultiCarriermodule.xSetCarrierForJoggingFromVis
        OnMouseClick: execute { SR_MultiCarrierModule.udiJoggingCarrierNr := 44; }
    Button (214,391 25x25), "45", colour toggle: SR_MultiCarrierModule.aifVisFeedback[45].ifFeedbackJogging.xJogActivated, invisible if: SR_MulticarrierModule.ifMulticarrier.ifFeedback.ifFeedbackConfiguration.udiNumberOfCarriers < 45, input disabled if: NOT SR_MainMachine.xActManual
        toggle SR_MultiCarriermodule.xSetCarrierForJoggingFromVis
        OnMouseClick: execute { SR_MultiCarrierModule.udiJoggingCarrierNr := 45; }
    Button (254,391 25x25), "46", colour toggle: SR_MultiCarrierModule.aifVisFeedback[46].ifFeedbackJogging.xJogActivated, invisible if: SR_MulticarrierModule.ifMulticarrier.ifFeedback.ifFeedbackConfiguration.udiNumberOfCarriers < 46, input disabled if: NOT SR_MainMachine.xActManual
        toggle SR_MultiCarriermodule.xSetCarrierForJoggingFromVis
        OnMouseClick: execute { SR_MultiCarrierModule.udiJoggingCarrierNr := 46; }
    Button (294,391 25x25), "47", colour toggle: SR_MultiCarrierModule.aifVisFeedback[47].ifFeedbackJogging.xJogActivated, invisible if: SR_MulticarrierModule.ifMulticarrier.ifFeedback.ifFeedbackConfiguration.udiNumberOfCarriers < 47, input disabled if: NOT SR_MainMachine.xActManual
        toggle SR_MultiCarriermodule.xSetCarrierForJoggingFromVis
        OnMouseClick: execute { SR_MultiCarrierModule.udiJoggingCarrierNr := 47; }
    Button (334,391 25x25), "48", colour toggle: SR_MultiCarrierModule.aifVisFeedback[48].ifFeedbackJogging.xJogActivated, invisible if: SR_MulticarrierModule.ifMulticarrier.ifFeedback.ifFeedbackConfiguration.udiNumberOfCarriers < 48, input disabled if: NOT SR_MainMachine.xActManual
        toggle SR_MultiCarriermodule.xSetCarrierForJoggingFromVis
        OnMouseClick: execute { SR_MultiCarrierModule.udiJoggingCarrierNr := 48; }
    Button (374,391 25x25), "49", colour toggle: SR_MultiCarrierModule.aifVisFeedback[49].ifFeedbackJogging.xJogActivated, invisible if: SR_MulticarrierModule.ifMulticarrier.ifFeedback.ifFeedbackConfiguration.udiNumberOfCarriers < 49, input disabled if: NOT SR_MainMachine.xActManual
        toggle SR_MultiCarriermodule.xSetCarrierForJoggingFromVis
        OnMouseClick: execute { SR_MultiCarrierModule.udiJoggingCarrierNr := 49; }
    Button (54,431 25x25), "51", colour toggle: SR_MultiCarrierModule.aifVisFeedback[51].ifFeedbackJogging.xJogActivated, invisible if: SR_MulticarrierModule.ifMulticarrier.ifFeedback.ifFeedbackConfiguration.udiNumberOfCarriers < 51, input disabled if: NOT SR_MainMachine.xActManual
        toggle SR_MultiCarriermodule.xSetCarrierForJoggingFromVis
        OnMouseClick: execute { SR_MultiCarrierModule.udiJoggingCarrierNr := 51; }
    Button (94,431 25x25), "52", colour toggle: SR_MultiCarrierModule.aifVisFeedback[52].ifFeedbackJogging.xJogActivated, invisible if: SR_MulticarrierModule.ifMulticarrier.ifFeedback.ifFeedbackConfiguration.udiNumberOfCarriers < 52, input disabled if: NOT SR_MainMachine.xActManual
        toggle SR_MultiCarriermodule.xSetCarrierForJoggingFromVis
        OnMouseClick: execute { SR_MultiCarrierModule.udiJoggingCarrierNr := 52; }
    Button (134,431 25x25), "53", colour toggle: SR_MultiCarrierModule.aifVisFeedback[53].ifFeedbackJogging.xJogActivated, invisible if: SR_MulticarrierModule.ifMulticarrier.ifFeedback.ifFeedbackConfiguration.udiNumberOfCarriers < 53, input disabled if: NOT SR_MainMachine.xActManual
        toggle SR_MultiCarriermodule.xSetCarrierForJoggingFromVis
        OnMouseClick: execute { SR_MultiCarrierModule.udiJoggingCarrierNr := 53; }
    Button (174,431 25x25), "54", colour toggle: SR_MultiCarrierModule.aifVisFeedback[54].ifFeedbackJogging.xJogActivated, invisible if: SR_MulticarrierModule.ifMulticarrier.ifFeedback.ifFeedbackConfiguration.udiNumberOfCarriers < 54, input disabled if: NOT SR_MainMachine.xActManual
        toggle SR_MultiCarriermodule.xSetCarrierForJoggingFromVis
        OnMouseClick: execute { SR_MultiCarrierModule.udiJoggingCarrierNr := 54; }
    Button (214,431 25x25), "55", colour toggle: SR_MultiCarrierModule.aifVisFeedback[55].ifFeedbackJogging.xJogActivated, invisible if: SR_MulticarrierModule.ifMulticarrier.ifFeedback.ifFeedbackConfiguration.udiNumberOfCarriers < 55, input disabled if: NOT SR_MainMachine.xActManual
        toggle SR_MultiCarriermodule.xSetCarrierForJoggingFromVis
        OnMouseClick: execute { SR_MultiCarrierModule.udiJoggingCarrierNr := 55; }
    Button (254,431 25x25), "56", colour toggle: SR_MultiCarrierModule.aifVisFeedback[56].ifFeedbackJogging.xJogActivated, invisible if: SR_MulticarrierModule.ifMulticarrier.ifFeedback.ifFeedbackConfiguration.udiNumberOfCarriers < 56, input disabled if: NOT SR_MainMachine.xActManual
        toggle SR_MultiCarriermodule.xSetCarrierForJoggingFromVis
        OnMouseClick: execute { SR_MultiCarrierModule.udiJoggingCarrierNr := 56; }
    Button (294,431 25x25), "57", colour toggle: SR_MultiCarrierModule.aifVisFeedback[57].ifFeedbackJogging.xJogActivated, invisible if: SR_MulticarrierModule.ifMulticarrier.ifFeedback.ifFeedbackConfiguration.udiNumberOfCarriers < 57, input disabled if: NOT SR_MainMachine.xActManual
        toggle SR_MultiCarriermodule.xSetCarrierForJoggingFromVis
        OnMouseClick: execute { SR_MultiCarrierModule.udiJoggingCarrierNr := 57; }
    Button (334,431 25x25), "58", colour toggle: SR_MultiCarrierModule.aifVisFeedback[58].ifFeedbackJogging.xJogActivated, invisible if: SR_MulticarrierModule.ifMulticarrier.ifFeedback.ifFeedbackConfiguration.udiNumberOfCarriers < 58, input disabled if: NOT SR_MainMachine.xActManual
        toggle SR_MultiCarriermodule.xSetCarrierForJoggingFromVis
        OnMouseClick: execute { SR_MultiCarrierModule.udiJoggingCarrierNr := 58; }
    Button (374,431 25x25), "59", colour toggle: SR_MultiCarrierModule.aifVisFeedback[59].ifFeedbackJogging.xJogActivated, invisible if: SR_MulticarrierModule.ifMulticarrier.ifFeedback.ifFeedbackConfiguration.udiNumberOfCarriers < 59, input disabled if: NOT SR_MainMachine.xActManual
        toggle SR_MultiCarriermodule.xSetCarrierForJoggingFromVis
        OnMouseClick: execute { SR_MultiCarrierModule.udiJoggingCarrierNr := 59; }
    Button (414,511 25x25), "80", colour toggle: SR_MultiCarrierModule.aifVisFeedback[80].ifFeedbackJogging.xJogActivated, invisible if: SR_MulticarrierModule.ifMulticarrier.ifFeedback.ifFeedbackConfiguration.udiNumberOfCarriers < 80, input disabled if: NOT SR_MainMachine.xActManual
        toggle SR_MultiCarriermodule.xSetCarrierForJoggingFromVis
        OnMouseClick: execute { SR_MultiCarrierModule.udiJoggingCarrierNr := 80; }
    Button (54,551 25x25), "81", colour toggle: SR_MultiCarrierModule.aifVisFeedback[81].ifFeedbackJogging.xJogActivated, invisible if: SR_MulticarrierModule.ifMulticarrier.ifFeedback.ifFeedbackConfiguration.udiNumberOfCarriers < 81, input disabled if: NOT SR_MainMachine.xActManual
        toggle SR_MultiCarriermodule.xSetCarrierForJoggingFromVis
        OnMouseClick: execute { SR_MultiCarrierModule.udiJoggingCarrierNr := 81; }
    Button (94,551 25x25), "82", colour toggle: SR_MultiCarrierModule.aifVisFeedback[82].ifFeedbackJogging.xJogActivated, invisible if: SR_MulticarrierModule.ifMulticarrier.ifFeedback.ifFeedbackConfiguration.udiNumberOfCarriers < 82, input disabled if: NOT SR_MainMachine.xActManual
        toggle SR_MultiCarriermodule.xSetCarrierForJoggingFromVis
        OnMouseClick: execute { SR_MultiCarrierModule.udiJoggingCarrierNr := 82; }
    Button (134,551 25x25), "83", colour toggle: SR_MultiCarrierModule.aifVisFeedback[83].ifFeedbackJogging.xJogActivated, invisible if: SR_MulticarrierModule.ifMulticarrier.ifFeedback.ifFeedbackConfiguration.udiNumberOfCarriers < 83, input disabled if: NOT SR_MainMachine.xActManual
        toggle SR_MultiCarriermodule.xSetCarrierForJoggingFromVis
        OnMouseClick: execute { SR_MultiCarrierModule.udiJoggingCarrierNr := 83; }
    Button (174,551 25x25), "84", colour toggle: SR_MultiCarrierModule.aifVisFeedback[84].ifFeedbackJogging.xJogActivated, invisible if: SR_MulticarrierModule.ifMulticarrier.ifFeedback.ifFeedbackConfiguration.udiNumberOfCarriers < 84, input disabled if: NOT SR_MainMachine.xActManual
        toggle SR_MultiCarriermodule.xSetCarrierForJoggingFromVis
        OnMouseClick: execute { SR_MultiCarrierModule.udiJoggingCarrierNr := 84; }
    Button (214,551 25x25), "85", colour toggle: SR_MultiCarrierModule.aifVisFeedback[85].ifFeedbackJogging.xJogActivated, invisible if: SR_MulticarrierModule.ifMulticarrier.ifFeedback.ifFeedbackConfiguration.udiNumberOfCarriers < 85, input disabled if: NOT SR_MainMachine.xActManual
        toggle SR_MultiCarriermodule.xSetCarrierForJoggingFromVis
        OnMouseClick: execute { SR_MultiCarrierModule.udiJoggingCarrierNr := 85; }
    Button (254,551 25x25), "88", colour toggle: SR_MultiCarrierModule.aifVisFeedback[88].ifFeedbackJogging.xJogActivated, invisible if: SR_MulticarrierModule.ifMulticarrier.ifFeedback.ifFeedbackConfiguration.udiNumberOfCarriers < 88, input disabled if: NOT SR_MainMachine.xActManual
        toggle SR_MultiCarriermodule.xSetCarrierForJoggingFromVis
        OnMouseClick: execute { SR_MultiCarrierModule.udiJoggingCarrierNr := 88; }
    Button (294,551 25x25), "87", colour toggle: SR_MultiCarrierModule.aifVisFeedback[87].ifFeedbackJogging.xJogActivated, invisible if: SR_MulticarrierModule.ifMulticarrier.ifFeedback.ifFeedbackConfiguration.udiNumberOfCarriers < 87, input disabled if: NOT SR_MainMachine.xActManual
        toggle SR_MultiCarriermodule.xSetCarrierForJoggingFromVis
        OnMouseClick: execute { SR_MultiCarrierModule.udiJoggingCarrierNr := 87; }
    Button (334,551 25x25), "88", colour toggle: SR_MultiCarrierModule.aifVisFeedback[88].ifFeedbackJogging.xJogActivated, invisible if: SR_MulticarrierModule.ifMulticarrier.ifFeedback.ifFeedbackConfiguration.udiNumberOfCarriers < 88, input disabled if: NOT SR_MainMachine.xActManual
        toggle SR_MultiCarriermodule.xSetCarrierForJoggingFromVis
        OnMouseClick: execute { SR_MultiCarrierModule.udiJoggingCarrierNr := 88; }
    Button (374,551 25x25), "89", colour toggle: SR_MultiCarrierModule.aifVisFeedback[89].ifFeedbackJogging.xJogActivated, invisible if: SR_MulticarrierModule.ifMulticarrier.ifFeedback.ifFeedbackConfiguration.udiNumberOfCarriers < 89, input disabled if: NOT SR_MainMachine.xActManual
        toggle SR_MultiCarriermodule.xSetCarrierForJoggingFromVis
        OnMouseClick: execute { SR_MultiCarrierModule.udiJoggingCarrierNr := 89; }
    Button (54,511 25x25), "71", colour toggle: SR_MultiCarrierModule.aifVisFeedback[71].ifFeedbackJogging.xJogActivated, invisible if: SR_MulticarrierModule.ifMulticarrier.ifFeedback.ifFeedbackConfiguration.udiNumberOfCarriers < 71, input disabled if: NOT SR_MainMachine.xActManual
        toggle SR_MultiCarriermodule.xSetCarrierForJoggingFromVis
        OnMouseClick: execute { SR_MultiCarrierModule.udiJoggingCarrierNr := 71; }
    Button (94,511 25x25), "72", colour toggle: SR_MultiCarrierModule.aifVisFeedback[72].ifFeedbackJogging.xJogActivated, invisible if: SR_MulticarrierModule.ifMulticarrier.ifFeedback.ifFeedbackConfiguration.udiNumberOfCarriers < 72, input disabled if: NOT SR_MainMachine.xActManual
        toggle SR_MultiCarriermodule.xSetCarrierForJoggingFromVis
        OnMouseClick: execute { SR_MultiCarrierModule.udiJoggingCarrierNr := 72; }
    Button (134,511 25x25), "73", colour toggle: SR_MultiCarrierModule.aifVisFeedback[73].ifFeedbackJogging.xJogActivated, invisible if: SR_MulticarrierModule.ifMulticarrier.ifFeedback.ifFeedbackConfiguration.udiNumberOfCarriers < 73, input disabled if: NOT SR_MainMachine.xActManual
        toggle SR_MultiCarriermodule.xSetCarrierForJoggingFromVis
        OnMouseClick: execute { SR_MultiCarrierModule.udiJoggingCarrierNr := 73; }
    Button (174,511 25x25), "74", colour toggle: SR_MultiCarrierModule.aifVisFeedback[74].ifFeedbackJogging.xJogActivated, invisible if: SR_MulticarrierModule.ifMulticarrier.ifFeedback.ifFeedbackConfiguration.udiNumberOfCarriers < 74, input disabled if: NOT SR_MainMachine.xActManual
        toggle SR_MultiCarriermodule.xSetCarrierForJoggingFromVis
        OnMouseClick: execute { SR_MultiCarrierModule.udiJoggingCarrierNr := 74; }
    Button (214,511 25x25), "75", colour toggle: SR_MultiCarrierModule.aifVisFeedback[75].ifFeedbackJogging.xJogActivated, invisible if: SR_MulticarrierModule.ifMulticarrier.ifFeedback.ifFeedbackConfiguration.udiNumberOfCarriers < 75, input disabled if: NOT SR_MainMachine.xActManual
        toggle SR_MultiCarriermodule.xSetCarrierForJoggingFromVis
        OnMouseClick: execute { SR_MultiCarrierModule.udiJoggingCarrierNr := 75; }
    Button (254,511 25x25), "76", colour toggle: SR_MultiCarrierModule.aifVisFeedback[76].ifFeedbackJogging.xJogActivated, invisible if: SR_MulticarrierModule.ifMulticarrier.ifFeedback.ifFeedbackConfiguration.udiNumberOfCarriers < 76, input disabled if: NOT SR_MainMachine.xActManual
        toggle SR_MultiCarriermodule.xSetCarrierForJoggingFromVis
        OnMouseClick: execute { SR_MultiCarrierModule.udiJoggingCarrierNr := 76; }
    Button (294,511 25x25), "77", colour toggle: SR_MultiCarrierModule.aifVisFeedback[77].ifFeedbackJogging.xJogActivated, invisible if: SR_MulticarrierModule.ifMulticarrier.ifFeedback.ifFeedbackConfiguration.udiNumberOfCarriers < 77, input disabled if: NOT SR_MainMachine.xActManual
        toggle SR_MultiCarriermodule.xSetCarrierForJoggingFromVis
        OnMouseClick: execute { SR_MultiCarrierModule.udiJoggingCarrierNr := 77; }
    Button (334,511 25x25), "78", colour toggle: SR_MultiCarrierModule.aifVisFeedback[78].ifFeedbackJogging.xJogActivated, invisible if: SR_MulticarrierModule.ifMulticarrier.ifFeedback.ifFeedbackConfiguration.udiNumberOfCarriers < 78, input disabled if: NOT SR_MainMachine.xActManual
        toggle SR_MultiCarriermodule.xSetCarrierForJoggingFromVis
        OnMouseClick: execute { SR_MultiCarrierModule.udiJoggingCarrierNr := 78; }
    Button (374,511 25x25), "79", colour toggle: SR_MultiCarrierModule.aifVisFeedback[79].ifFeedbackJogging.xJogActivated, invisible if: SR_MulticarrierModule.ifMulticarrier.ifFeedback.ifFeedbackConfiguration.udiNumberOfCarriers < 79, input disabled if: NOT SR_MainMachine.xActManual
        toggle SR_MultiCarriermodule.xSetCarrierForJoggingFromVis
        OnMouseClick: execute { SR_MultiCarrierModule.udiJoggingCarrierNr := 79; }
    Button (414,551 25x25), "90", colour toggle: SR_MultiCarrierModule.aifVisFeedback[90].ifFeedbackJogging.xJogActivated, invisible if: SR_MulticarrierModule.ifMulticarrier.ifFeedback.ifFeedbackConfiguration.udiNumberOfCarriers < 90, input disabled if: NOT SR_MainMachine.xActManual
        toggle SR_MultiCarriermodule.xSetCarrierForJoggingFromVis
        OnMouseClick: execute { SR_MultiCarrierModule.udiJoggingCarrierNr := 90; }
    Button (54,591 25x25), "91", colour toggle: SR_MultiCarrierModule.aifVisFeedback[91].ifFeedbackJogging.xJogActivated, invisible if: SR_MulticarrierModule.ifMulticarrier.ifFeedback.ifFeedbackConfiguration.udiNumberOfCarriers < 91, input disabled if: NOT SR_MainMachine.xActManual
        toggle SR_MultiCarriermodule.xSetCarrierForJoggingFromVis
        OnMouseClick: execute { SR_MultiCarrierModule.udiJoggingCarrierNr := 91; }
    Button (94,591 25x25), "92", colour toggle: SR_MultiCarrierModule.aifVisFeedback[92].ifFeedbackJogging.xJogActivated, invisible if: SR_MulticarrierModule.ifMulticarrier.ifFeedback.ifFeedbackConfiguration.udiNumberOfCarriers < 92, input disabled if: NOT SR_MainMachine.xActManual
        toggle SR_MultiCarriermodule.xSetCarrierForJoggingFromVis
        OnMouseClick: execute { SR_MultiCarrierModule.udiJoggingCarrierNr := 92; }
    Button (134,591 25x25), "93", colour toggle: SR_MultiCarrierModule.aifVisFeedback[93].ifFeedbackJogging.xJogActivated, invisible if: SR_MulticarrierModule.ifMulticarrier.ifFeedback.ifFeedbackConfiguration.udiNumberOfCarriers < 93, input disabled if: NOT SR_MainMachine.xActManual
        toggle SR_MultiCarriermodule.xSetCarrierForJoggingFromVis
        OnMouseClick: execute { SR_MultiCarrierModule.udiJoggingCarrierNr := 93; }
    Button (174,591 25x25), "94", colour toggle: SR_MultiCarrierModule.aifVisFeedback[94].ifFeedbackJogging.xJogActivated, invisible if: SR_MulticarrierModule.ifMulticarrier.ifFeedback.ifFeedbackConfiguration.udiNumberOfCarriers < 94, input disabled if: NOT SR_MainMachine.xActManual
        toggle SR_MultiCarriermodule.xSetCarrierForJoggingFromVis
        OnMouseClick: execute { SR_MultiCarrierModule.udiJoggingCarrierNr := 94; }
    Button (214,591 25x25), "95", colour toggle: SR_MultiCarrierModule.aifVisFeedback[95].ifFeedbackJogging.xJogActivated, invisible if: SR_MulticarrierModule.ifMulticarrier.ifFeedback.ifFeedbackConfiguration.udiNumberOfCarriers < 95, input disabled if: NOT SR_MainMachine.xActManual
        toggle SR_MultiCarriermodule.xSetCarrierForJoggingFromVis
        OnMouseClick: execute { SR_MultiCarrierModule.udiJoggingCarrierNr := 95; }
    Button (254,591 25x25), "96", colour toggle: SR_MultiCarrierModule.aifVisFeedback[96].ifFeedbackJogging.xJogActivated, invisible if: SR_MulticarrierModule.ifMulticarrier.ifFeedback.ifFeedbackConfiguration.udiNumberOfCarriers < 96, input disabled if: NOT SR_MainMachine.xActManual
        toggle SR_MultiCarriermodule.xSetCarrierForJoggingFromVis
        OnMouseClick: execute { SR_MultiCarrierModule.udiJoggingCarrierNr := 96; }
    Button (294,591 25x25), "97", colour toggle: SR_MultiCarrierModule.aifVisFeedback[97].ifFeedbackJogging.xJogActivated, invisible if: SR_MulticarrierModule.ifMulticarrier.ifFeedback.ifFeedbackConfiguration.udiNumberOfCarriers < 97, input disabled if: NOT SR_MainMachine.xActManual
        toggle SR_MultiCarriermodule.xSetCarrierForJoggingFromVis
        OnMouseClick: execute { SR_MultiCarrierModule.udiJoggingCarrierNr := 97; }
    Button (334,591 25x25), "98", colour toggle: SR_MultiCarrierModule.aifVisFeedback[98].ifFeedbackJogging.xJogActivated, invisible if: SR_MulticarrierModule.ifMulticarrier.ifFeedback.ifFeedbackConfiguration.udiNumberOfCarriers < 98, input disabled if: NOT SR_MainMachine.xActManual
        toggle SR_MultiCarriermodule.xSetCarrierForJoggingFromVis
        OnMouseClick: execute { SR_MultiCarrierModule.udiJoggingCarrierNr := 98; }
    Button (374,591 25x25), "99", colour toggle: SR_MultiCarrierModule.aifVisFeedback[99].ifFeedbackJogging.xJogActivated, invisible if: SR_MulticarrierModule.ifMulticarrier.ifFeedback.ifFeedbackConfiguration.udiNumberOfCarriers < 99, input disabled if: NOT SR_MainMachine.xActManual
        toggle SR_MultiCarriermodule.xSetCarrierForJoggingFromVis
        OnMouseClick: execute { SR_MultiCarrierModule.udiJoggingCarrierNr := 99; }
    Button (414,591 25x25), "100", colour toggle: SR_MultiCarrierModule.aifVisFeedback[100].ifFeedbackJogging.xJogActivated, invisible if: SR_MulticarrierModule.ifMulticarrier.ifFeedback.ifFeedbackConfiguration.udiNumberOfCarriers < 100, input disabled if: NOT SR_MainMachine.xActManual
        toggle SR_MultiCarriermodule.xSetCarrierForJoggingFromVis
        OnMouseClick: execute { SR_MultiCarrierModule.udiJoggingCarrierNr := 100; }
    Button (54,631 25x25), "101", colour toggle: SR_MultiCarrierModule.aifVisFeedback[101].ifFeedbackJogging.xJogActivated, invisible if: SR_MulticarrierModule.ifMulticarrier.ifFeedback.ifFeedbackConfiguration.udiNumberOfCarriers < 101, input disabled if: NOT SR_MainMachine.xActManual
        toggle SR_MultiCarriermodule.xSetCarrierForJoggingFromVis
        OnMouseClick: execute { SR_MultiCarrierModule.udiJoggingCarrierNr := 101; }
    Button (94,631 25x25), "102", colour toggle: SR_MultiCarrierModule.aifVisFeedback[102].ifFeedbackJogging.xJogActivated, invisible if: SR_MulticarrierModule.ifMulticarrier.ifFeedback.ifFeedbackConfiguration.udiNumberOfCarriers < 102, input disabled if: NOT SR_MainMachine.xActManual
        toggle SR_MultiCarriermodule.xSetCarrierForJoggingFromVis
        OnMouseClick: execute { SR_MultiCarrierModule.udiJoggingCarrierNr := 102; }
    Button (134,631 25x25), "103", colour toggle: SR_MultiCarrierModule.aifVisFeedback[103].ifFeedbackJogging.xJogActivated, invisible if: SR_MulticarrierModule.ifMulticarrier.ifFeedback.ifFeedbackConfiguration.udiNumberOfCarriers < 103, input disabled if: NOT SR_MainMachine.xActManual
        toggle SR_MultiCarriermodule.xSetCarrierForJoggingFromVis
        OnMouseClick: execute { SR_MultiCarrierModule.udiJoggingCarrierNr := 103; }
    Button (174,631 25x25), "104", colour toggle: SR_MultiCarrierModule.aifVisFeedback[104].ifFeedbackJogging.xJogActivated, invisible if: SR_MulticarrierModule.ifMulticarrier.ifFeedback.ifFeedbackConfiguration.udiNumberOfCarriers < 104, input disabled if: NOT SR_MainMachine.xActManual
        toggle SR_MultiCarriermodule.xSetCarrierForJoggingFromVis
        OnMouseClick: execute { SR_MultiCarrierModule.udiJoggingCarrierNr := 104; }
    Button (214,631 25x25), "105", colour toggle: SR_MultiCarrierModule.aifVisFeedback[105].ifFeedbackJogging.xJogActivated, invisible if: SR_MulticarrierModule.ifMulticarrier.ifFeedback.ifFeedbackConfiguration.udiNumberOfCarriers < 105, input disabled if: NOT SR_MainMachine.xActManual
        toggle SR_MultiCarriermodule.xSetCarrierForJoggingFromVis
        OnMouseClick: execute { SR_MultiCarrierModule.udiJoggingCarrierNr := 105; }
    Button (254,631 25x25), "106", colour toggle: SR_MultiCarrierModule.aifVisFeedback[106].ifFeedbackJogging.xJogActivated, invisible if: SR_MulticarrierModule.ifMulticarrier.ifFeedback.ifFeedbackConfiguration.udiNumberOfCarriers < 106, input disabled if: NOT SR_MainMachine.xActManual
        toggle SR_MultiCarriermodule.xSetCarrierForJoggingFromVis
        OnMouseClick: execute { SR_MultiCarrierModule.udiJoggingCarrierNr := 106; }
    Button (294,631 25x25), "107", colour toggle: SR_MultiCarrierModule.aifVisFeedback[107].ifFeedbackJogging.xJogActivated, invisible if: SR_MulticarrierModule.ifMulticarrier.ifFeedback.ifFeedbackConfiguration.udiNumberOfCarriers < 107, input disabled if: NOT SR_MainMachine.xActManual
        toggle SR_MultiCarriermodule.xSetCarrierForJoggingFromVis
        OnMouseClick: execute { SR_MultiCarrierModule.udiJoggingCarrierNr := 107; }
    Button (334,631 25x25), "108", colour toggle: SR_MultiCarrierModule.aifVisFeedback[108].ifFeedbackJogging.xJogActivated, invisible if: SR_MulticarrierModule.ifMulticarrier.ifFeedback.ifFeedbackConfiguration.udiNumberOfCarriers < 108, input disabled if: NOT SR_MainMachine.xActManual
        toggle SR_MultiCarriermodule.xSetCarrierForJoggingFromVis
        OnMouseClick: execute { SR_MultiCarrierModule.udiJoggingCarrierNr := 108; }
    Button (374,631 25x25), "109", colour toggle: SR_MultiCarrierModule.aifVisFeedback[109].ifFeedbackJogging.xJogActivated, invisible if: SR_MulticarrierModule.ifMulticarrier.ifFeedback.ifFeedbackConfiguration.udiNumberOfCarriers < 109, input disabled if: NOT SR_MainMachine.xActManual
        toggle SR_MultiCarriermodule.xSetCarrierForJoggingFromVis
        OnMouseClick: execute { SR_MultiCarrierModule.udiJoggingCarrierNr := 109; }
    Button (414,631 25x25), "110", colour toggle: SR_MultiCarrierModule.aifVisFeedback[110].ifFeedbackJogging.xJogActivated, invisible if: SR_MulticarrierModule.ifMulticarrier.ifFeedback.ifFeedbackConfiguration.udiNumberOfCarriers < 110, input disabled if: NOT SR_MainMachine.xActManual
        toggle SR_MultiCarriermodule.xSetCarrierForJoggingFromVis
        OnMouseClick: execute { SR_MultiCarrierModule.udiJoggingCarrierNr := 110; }
    Button (54,671 25x25), "111", colour toggle: SR_MultiCarrierModule.aifVisFeedback[111].ifFeedbackJogging.xJogActivated, invisible if: SR_MulticarrierModule.ifMulticarrier.ifFeedback.ifFeedbackConfiguration.udiNumberOfCarriers < 111, input disabled if: NOT SR_MainMachine.xActManual
        toggle SR_MultiCarriermodule.xSetCarrierForJoggingFromVis
        OnMouseClick: execute { SR_MultiCarrierModule.udiJoggingCarrierNr := 111; }
    Button (94,671 25x25), "112", colour toggle: SR_MultiCarrierModule.aifVisFeedback[112].ifFeedbackJogging.xJogActivated, invisible if: SR_MulticarrierModule.ifMulticarrier.ifFeedback.ifFeedbackConfiguration.udiNumberOfCarriers < 112, input disabled if: NOT SR_MainMachine.xActManual
        toggle SR_MultiCarriermodule.xSetCarrierForJoggingFromVis
        OnMouseClick: execute { SR_MultiCarrierModule.udiJoggingCarrierNr := 112; }
    Button (134,671 25x25), "113", colour toggle: SR_MultiCarrierModule.aifVisFeedback[113].ifFeedbackJogging.xJogActivated, invisible if: SR_MulticarrierModule.ifMulticarrier.ifFeedback.ifFeedbackConfiguration.udiNumberOfCarriers < 113, input disabled if: NOT SR_MainMachine.xActManual
        toggle SR_MultiCarriermodule.xSetCarrierForJoggingFromVis
        OnMouseClick: execute { SR_MultiCarrierModule.udiJoggingCarrierNr := 113; }
    Button (174,671 25x25), "114", colour toggle: SR_MultiCarrierModule.aifVisFeedback[114].ifFeedbackJogging.xJogActivated, invisible if: SR_MulticarrierModule.ifMulticarrier.ifFeedback.ifFeedbackConfiguration.udiNumberOfCarriers < 114, input disabled if: NOT SR_MainMachine.xActManual
        toggle SR_MultiCarriermodule.xSetCarrierForJoggingFromVis
        OnMouseClick: execute { SR_MultiCarrierModule.udiJoggingCarrierNr := 114; }
    Button (214,671 25x25), "115", colour toggle: SR_MultiCarrierModule.aifVisFeedback[115].ifFeedbackJogging.xJogActivated, invisible if: SR_MulticarrierModule.ifMulticarrier.ifFeedback.ifFeedbackConfiguration.udiNumberOfCarriers < 115, input disabled if: NOT SR_MainMachine.xActManual
        toggle SR_MultiCarriermodule.xSetCarrierForJoggingFromVis
        OnMouseClick: execute { SR_MultiCarrierModule.udiJoggingCarrierNr := 115; }
    Button (254,671 25x25), "116", colour toggle: SR_MultiCarrierModule.aifVisFeedback[116].ifFeedbackJogging.xJogActivated, invisible if: SR_MulticarrierModule.ifMulticarrier.ifFeedback.ifFeedbackConfiguration.udiNumberOfCarriers < 116, input disabled if: NOT SR_MainMachine.xActManual
        toggle SR_MultiCarriermodule.xSetCarrierForJoggingFromVis
        OnMouseClick: execute { SR_MultiCarrierModule.udiJoggingCarrierNr := 116; }
    Button (294,671 25x25), "117", colour toggle: SR_MultiCarrierModule.aifVisFeedback[117].ifFeedbackJogging.xJogActivated, invisible if: SR_MulticarrierModule.ifMulticarrier.ifFeedback.ifFeedbackConfiguration.udiNumberOfCarriers < 117, input disabled if: NOT SR_MainMachine.xActManual
        toggle SR_MultiCarriermodule.xSetCarrierForJoggingFromVis
        OnMouseClick: execute { SR_MultiCarrierModule.udiJoggingCarrierNr := 117; }
    Button (334,671 25x25), "118", colour toggle: SR_MultiCarrierModule.aifVisFeedback[118].ifFeedbackJogging.xJogActivated, invisible if: SR_MulticarrierModule.ifMulticarrier.ifFeedback.ifFeedbackConfiguration.udiNumberOfCarriers < 118, input disabled if: NOT SR_MainMachine.xActManual
        toggle SR_MultiCarriermodule.xSetCarrierForJoggingFromVis
        OnMouseClick: execute { SR_MultiCarrierModule.udiJoggingCarrierNr := 118; }
    Button (374,671 25x25), "119", colour toggle: SR_MultiCarrierModule.aifVisFeedback[119].ifFeedbackJogging.xJogActivated, invisible if: SR_MulticarrierModule.ifMulticarrier.ifFeedback.ifFeedbackConfiguration.udiNumberOfCarriers < 119, input disabled if: NOT SR_MainMachine.xActManual
        toggle SR_MultiCarriermodule.xSetCarrierForJoggingFromVis
        OnMouseClick: execute { SR_MultiCarrierModule.udiJoggingCarrierNr := 119; }
    Button (414,671 25x25), "120", colour toggle: SR_MultiCarrierModule.aifVisFeedback[120].ifFeedbackJogging.xJogActivated, invisible if: SR_MulticarrierModule.ifMulticarrier.ifFeedback.ifFeedbackConfiguration.udiNumberOfCarriers < 120, input disabled if: NOT SR_MainMachine.xActManual
        toggle SR_MultiCarriermodule.xSetCarrierForJoggingFromVis
        OnMouseClick: execute { SR_MultiCarrierModule.udiJoggingCarrierNr := 120; }
    Button (54,711 25x25), "121", colour toggle: SR_MultiCarrierModule.aifVisFeedback[121].ifFeedbackJogging.xJogActivated, invisible if: SR_MulticarrierModule.ifMulticarrier.ifFeedback.ifFeedbackConfiguration.udiNumberOfCarriers < 121, input disabled if: NOT SR_MainMachine.xActManual
        toggle SR_MultiCarriermodule.xSetCarrierForJoggingFromVis
        OnMouseClick: execute { SR_MultiCarrierModule.udiJoggingCarrierNr := 121; }
    Button (94,711 25x25), "122", colour toggle: SR_MultiCarrierModule.aifVisFeedback[122].ifFeedbackJogging.xJogActivated, invisible if: SR_MulticarrierModule.ifMulticarrier.ifFeedback.ifFeedbackConfiguration.udiNumberOfCarriers < 122, input disabled if: NOT SR_MainMachine.xActManual
        toggle SR_MultiCarriermodule.xSetCarrierForJoggingFromVis
        OnMouseClick: execute { SR_MultiCarrierModule.udiJoggingCarrierNr := 122; }
    Button (134,711 25x25), "123", colour toggle: SR_MultiCarrierModule.aifVisFeedback[123].ifFeedbackJogging.xJogActivated, invisible if: SR_MulticarrierModule.ifMulticarrier.ifFeedback.ifFeedbackConfiguration.udiNumberOfCarriers < 123, input disabled if: NOT SR_MainMachine.xActManual
        toggle SR_MultiCarriermodule.xSetCarrierForJoggingFromVis
        OnMouseClick: execute { SR_MultiCarrierModule.udiJoggingCarrierNr := 123; }
    Button (174,711 25x25), "124", colour toggle: SR_MultiCarrierModule.aifVisFeedback[124].ifFeedbackJogging.xJogActivated, invisible if: SR_MulticarrierModule.ifMulticarrier.ifFeedback.ifFeedbackConfiguration.udiNumberOfCarriers < 124, input disabled if: NOT SR_MainMachine.xActManual
        toggle SR_MultiCarriermodule.xSetCarrierForJoggingFromVis
        OnMouseClick: execute { SR_MultiCarrierModule.udiJoggingCarrierNr := 124; }
    Button (214,711 25x25), "125", colour toggle: SR_MultiCarrierModule.aifVisFeedback[125].ifFeedbackJogging.xJogActivated, invisible if: SR_MulticarrierModule.ifMulticarrier.ifFeedback.ifFeedbackConfiguration.udiNumberOfCarriers < 125, input disabled if: NOT SR_MainMachine.xActManual
        toggle SR_MultiCarriermodule.xSetCarrierForJoggingFromVis
        OnMouseClick: execute { SR_MultiCarrierModule.udiJoggingCarrierNr := 125; }
    Button (254,711 25x25), "126", colour toggle: SR_MultiCarrierModule.aifVisFeedback[126].ifFeedbackJogging.xJogActivated, invisible if: SR_MulticarrierModule.ifMulticarrier.ifFeedback.ifFeedbackConfiguration.udiNumberOfCarriers < 126, input disabled if: NOT SR_MainMachine.xActManual
        toggle SR_MultiCarriermodule.xSetCarrierForJoggingFromVis
        OnMouseClick: execute { SR_MultiCarrierModule.udiJoggingCarrierNr := 126; }
    Button (294,711 25x25), "127", colour toggle: SR_MultiCarrierModule.aifVisFeedback[127].ifFeedbackJogging.xJogActivated, invisible if: SR_MulticarrierModule.ifMulticarrier.ifFeedback.ifFeedbackConfiguration.udiNumberOfCarriers < 127, input disabled if: NOT SR_MainMachine.xActManual
        toggle SR_MultiCarriermodule.xSetCarrierForJoggingFromVis
        OnMouseClick: execute { SR_MultiCarrierModule.udiJoggingCarrierNr := 127; }
    Button (334,711 25x25), "128", colour toggle: SR_MultiCarrierModule.aifVisFeedback[128].ifFeedbackJogging.xJogActivated, invisible if: SR_MulticarrierModule.ifMulticarrier.ifFeedback.ifFeedbackConfiguration.udiNumberOfCarriers < 128, input disabled if: NOT SR_MainMachine.xActManual
        toggle SR_MultiCarriermodule.xSetCarrierForJoggingFromVis
        OnMouseClick: execute { SR_MultiCarrierModule.udiJoggingCarrierNr := 128; }
    Button (374,711 25x25), "129", colour toggle: SR_MultiCarrierModule.aifVisFeedback[129].ifFeedbackJogging.xJogActivated, invisible if: SR_MulticarrierModule.ifMulticarrier.ifFeedback.ifFeedbackConfiguration.udiNumberOfCarriers < 129, input disabled if: NOT SR_MainMachine.xActManual
        toggle SR_MultiCarriermodule.xSetCarrierForJoggingFromVis
        OnMouseClick: execute { SR_MultiCarrierModule.udiJoggingCarrierNr := 129; }
    Button (414,711 25x25), "130", colour toggle: SR_MultiCarrierModule.aifVisFeedback[130].ifFeedbackJogging.xJogActivated, invisible if: SR_MulticarrierModule.ifMulticarrier.ifFeedback.ifFeedbackConfiguration.udiNumberOfCarriers < 130, input disabled if: NOT SR_MainMachine.xActManual
        toggle SR_MultiCarriermodule.xSetCarrierForJoggingFromVis
        OnMouseClick: execute { SR_MultiCarrierModule.udiJoggingCarrierNr := 130; }
    Button (54,751 25x25), "131", colour toggle: SR_MultiCarrierModule.aifVisFeedback[131].ifFeedbackJogging.xJogActivated, invisible if: SR_MulticarrierModule.ifMulticarrier.ifFeedback.ifFeedbackConfiguration.udiNumberOfCarriers < 131, input disabled if: NOT SR_MainMachine.xActManual
        toggle SR_MultiCarriermodule.xSetCarrierForJoggingFromVis
        OnMouseClick: execute { SR_MultiCarrierModule.udiJoggingCarrierNr := 131; }
    Button (94,751 25x25), "132", colour toggle: SR_MultiCarrierModule.aifVisFeedback[132].ifFeedbackJogging.xJogActivated, invisible if: SR_MulticarrierModule.ifMulticarrier.ifFeedback.ifFeedbackConfiguration.udiNumberOfCarriers < 132, input disabled if: NOT SR_MainMachine.xActManual
        toggle SR_MultiCarriermodule.xSetCarrierForJoggingFromVis
        OnMouseClick: execute { SR_MultiCarrierModule.udiJoggingCarrierNr := 132; }
    Button (134,751 25x25), "133", colour toggle: SR_MultiCarrierModule.aifVisFeedback[133].ifFeedbackJogging.xJogActivated, invisible if: SR_MulticarrierModule.ifMulticarrier.ifFeedback.ifFeedbackConfiguration.udiNumberOfCarriers < 133, input disabled if: NOT SR_MainMachine.xActManual
        toggle SR_MultiCarriermodule.xSetCarrierForJoggingFromVis
        OnMouseClick: execute { SR_MultiCarrierModule.udiJoggingCarrierNr := 133; }
    Button (174,751 25x25), "134", colour toggle: SR_MultiCarrierModule.aifVisFeedback[134].ifFeedbackJogging.xJogActivated, invisible if: SR_MulticarrierModule.ifMulticarrier.ifFeedback.ifFeedbackConfiguration.udiNumberOfCarriers < 134, input disabled if: NOT SR_MainMachine.xActManual
        toggle SR_MultiCarriermodule.xSetCarrierForJoggingFromVis
        OnMouseClick: execute { SR_MultiCarrierModule.udiJoggingCarrierNr := 134; }
    Button (214,751 25x25), "135", colour toggle: SR_MultiCarrierModule.aifVisFeedback[135].ifFeedbackJogging.xJogActivated, invisible if: SR_MulticarrierModule.ifMulticarrier.ifFeedback.ifFeedbackConfiguration.udiNumberOfCarriers < 135, input disabled if: NOT SR_MainMachine.xActManual
        toggle SR_MultiCarriermodule.xSetCarrierForJoggingFromVis
        OnMouseClick: execute { SR_MultiCarrierModule.udiJoggingCarrierNr := 135; }
    Button (254,751 25x25), "136", colour toggle: SR_MultiCarrierModule.aifVisFeedback[136].ifFeedbackJogging.xJogActivated, invisible if: SR_MulticarrierModule.ifMulticarrier.ifFeedback.ifFeedbackConfiguration.udiNumberOfCarriers < 136, input disabled if: NOT SR_MainMachine.xActManual
        toggle SR_MultiCarriermodule.xSetCarrierForJoggingFromVis
        OnMouseClick: execute { SR_MultiCarrierModule.udiJoggingCarrierNr := 136; }
    Button (294,751 25x25), "137", colour toggle: SR_MultiCarrierModule.aifVisFeedback[137].ifFeedbackJogging.xJogActivated, invisible if: SR_MulticarrierModule.ifMulticarrier.ifFeedback.ifFeedbackConfiguration.udiNumberOfCarriers < 137, input disabled if: NOT SR_MainMachine.xActManual
        toggle SR_MultiCarriermodule.xSetCarrierForJoggingFromVis
        OnMouseClick: execute { SR_MultiCarrierModule.udiJoggingCarrierNr := 137; }
    Button (334,751 25x25), "138", colour toggle: SR_MultiCarrierModule.aifVisFeedback[138].ifFeedbackJogging.xJogActivated, invisible if: SR_MulticarrierModule.ifMulticarrier.ifFeedback.ifFeedbackConfiguration.udiNumberOfCarriers < 138, input disabled if: NOT SR_MainMachine.xActManual
        toggle SR_MultiCarriermodule.xSetCarrierForJoggingFromVis
        OnMouseClick: execute { SR_MultiCarrierModule.udiJoggingCarrierNr := 138; }
    Button (374,751 25x25), "139", colour toggle: SR_MultiCarrierModule.aifVisFeedback[139].ifFeedbackJogging.xJogActivated, invisible if: SR_MulticarrierModule.ifMulticarrier.ifFeedback.ifFeedbackConfiguration.udiNumberOfCarriers < 139, input disabled if: NOT SR_MainMachine.xActManual
        toggle SR_MultiCarriermodule.xSetCarrierForJoggingFromVis
        OnMouseClick: execute { SR_MultiCarrierModule.udiJoggingCarrierNr := 139; }
    Button (414,751 25x25), "140", colour toggle: SR_MultiCarrierModule.aifVisFeedback[140].ifFeedbackJogging.xJogActivated, invisible if: SR_MulticarrierModule.ifMulticarrier.ifFeedback.ifFeedbackConfiguration.udiNumberOfCarriers < 140, input disabled if: NOT SR_MainMachine.xActManual
        toggle SR_MultiCarriermodule.xSetCarrierForJoggingFromVis
        OnMouseClick: execute { SR_MultiCarrierModule.udiJoggingCarrierNr := 140; }
    Button (54,791 25x25), "141", colour toggle: SR_MultiCarrierModule.aifVisFeedback[141].ifFeedbackJogging.xJogActivated, invisible if: SR_MulticarrierModule.ifMulticarrier.ifFeedback.ifFeedbackConfiguration.udiNumberOfCarriers < 141, input disabled if: NOT SR_MainMachine.xActManual
        toggle SR_MultiCarriermodule.xSetCarrierForJoggingFromVis
        OnMouseClick: execute { SR_MultiCarrierModule.udiJoggingCarrierNr := 141; }
    Button (94,791 25x25), "142", colour toggle: SR_MultiCarrierModule.aifVisFeedback[142].ifFeedbackJogging.xJogActivated, invisible if: SR_MulticarrierModule.ifMulticarrier.ifFeedback.ifFeedbackConfiguration.udiNumberOfCarriers < 142, input disabled if: NOT SR_MainMachine.xActManual
        toggle SR_MultiCarriermodule.xSetCarrierForJoggingFromVis
        OnMouseClick: execute { SR_MultiCarrierModule.udiJoggingCarrierNr := 142; }
    Button (134,791 25x25), "143", colour toggle: SR_MultiCarrierModule.aifVisFeedback[143].ifFeedbackJogging.xJogActivated, invisible if: SR_MulticarrierModule.ifMulticarrier.ifFeedback.ifFeedbackConfiguration.udiNumberOfCarriers < 143, input disabled if: NOT SR_MainMachine.xActManual
        toggle SR_MultiCarriermodule.xSetCarrierForJoggingFromVis
        OnMouseClick: execute { SR_MultiCarrierModule.udiJoggingCarrierNr := 143; }
    Button (174,791 25x25), "144", colour toggle: SR_MultiCarrierModule.aifVisFeedback[144].ifFeedbackJogging.xJogActivated, invisible if: SR_MulticarrierModule.ifMulticarrier.ifFeedback.ifFeedbackConfiguration.udiNumberOfCarriers < 144, input disabled if: NOT SR_MainMachine.xActManual
        toggle SR_MultiCarriermodule.xSetCarrierForJoggingFromVis
        OnMouseClick: execute { SR_MultiCarrierModule.udiJoggingCarrierNr := 144; }
    Button (214,791 25x25), "145", colour toggle: SR_MultiCarrierModule.aifVisFeedback[145].ifFeedbackJogging.xJogActivated, invisible if: SR_MulticarrierModule.ifMulticarrier.ifFeedback.ifFeedbackConfiguration.udiNumberOfCarriers < 145, input disabled if: NOT SR_MainMachine.xActManual
        toggle SR_MultiCarriermodule.xSetCarrierForJoggingFromVis
        OnMouseClick: execute { SR_MultiCarrierModule.udiJoggingCarrierNr := 145; }
    Button (254,791 25x25), "146", colour toggle: SR_MultiCarrierModule.aifVisFeedback[146].ifFeedbackJogging.xJogActivated, invisible if: SR_MulticarrierModule.ifMulticarrier.ifFeedback.ifFeedbackConfiguration.udiNumberOfCarriers < 146, input disabled if: NOT SR_MainMachine.xActManual
        toggle SR_MultiCarriermodule.xSetCarrierForJoggingFromVis
        OnMouseClick: execute { SR_MultiCarrierModule.udiJoggingCarrierNr := 146; }
    Button (294,791 25x25), "147", colour toggle: SR_MultiCarrierModule.aifVisFeedback[147].ifFeedbackJogging.xJogActivated, invisible if: SR_MulticarrierModule.ifMulticarrier.ifFeedback.ifFeedbackConfiguration.udiNumberOfCarriers < 147, input disabled if: NOT SR_MainMachine.xActManual
        toggle SR_MultiCarriermodule.xSetCarrierForJoggingFromVis
        OnMouseClick: execute { SR_MultiCarrierModule.udiJoggingCarrierNr := 147; }
    Button (334,791 25x25), "148", colour toggle: SR_MultiCarrierModule.aifVisFeedback[148].ifFeedbackJogging.xJogActivated, invisible if: SR_MulticarrierModule.ifMulticarrier.ifFeedback.ifFeedbackConfiguration.udiNumberOfCarriers < 148, input disabled if: NOT SR_MainMachine.xActManual
        toggle SR_MultiCarriermodule.xSetCarrierForJoggingFromVis
        OnMouseClick: execute { SR_MultiCarrierModule.udiJoggingCarrierNr := 148; }
    Button (374,791 25x25), "149", colour toggle: SR_MultiCarrierModule.aifVisFeedback[149].ifFeedbackJogging.xJogActivated, invisible if: SR_MulticarrierModule.ifMulticarrier.ifFeedback.ifFeedbackConfiguration.udiNumberOfCarriers < 149, input disabled if: NOT SR_MainMachine.xActManual
        toggle SR_MultiCarriermodule.xSetCarrierForJoggingFromVis
        OnMouseClick: execute { SR_MultiCarrierModule.udiJoggingCarrierNr := 149; }
    Button (414,791 25x25), "150", colour toggle: SR_MultiCarrierModule.aifVisFeedback[150].ifFeedbackJogging.xJogActivated, invisible if: SR_MulticarrierModule.ifMulticarrier.ifFeedback.ifFeedbackConfiguration.udiNumberOfCarriers < 150, input disabled if: NOT SR_MainMachine.xActManual
        toggle SR_MultiCarriermodule.xSetCarrierForJoggingFromVis
        OnMouseClick: execute { SR_MultiCarrierModule.udiJoggingCarrierNr := 150; }
END_VISUALIZATION

// LMC_PacDrive/Application/TemplateFullProgrammingFramework/Visualization/Multicarrier/Vis_NoOpMode
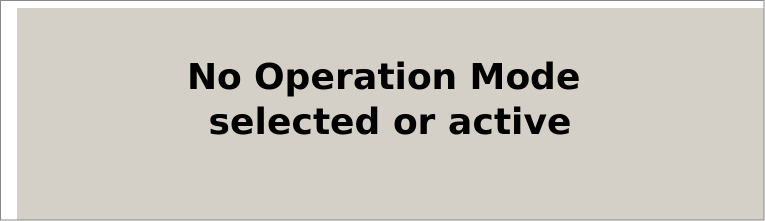
VISUALIZATION Vis_NoOpMode  // 765x221
    Rectangle (17,8 746x211), "No Operation Mode selected or active"
END_VISUALIZATION

// LMC_PacDrive/Application/TemplateFullProgrammingFramework/Visualization/Multicarrier/Vis_Positions
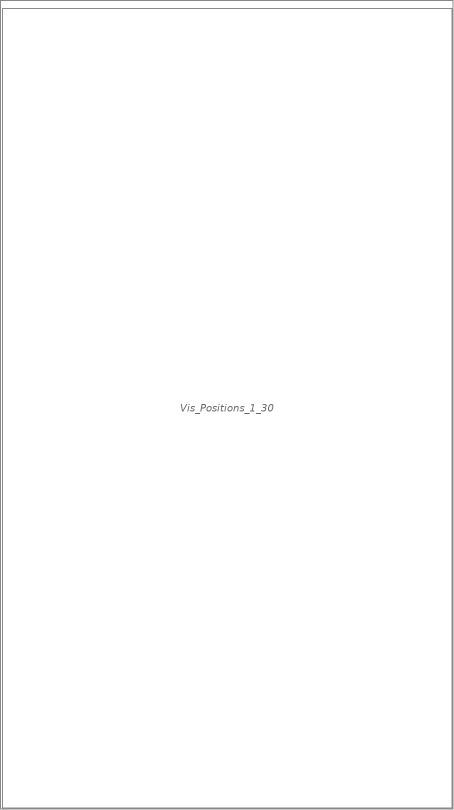
VISUALIZATION Vis_Positions  // 454x810
    TabControl (2,8 450x800)
        shows Vis_Positions_1_30()
        shows Vis_Positions_31_60()
        shows Vis_Positions_61_90()
        shows Vis_Positions_91_120()
        shows Vis_Positions_121_150()
        [0]: TabTitle=1-30
        [1]: TabTitle=31-60
        [2]: TabTitle=61-90
        [3]: TabTitle=91-120
        [4]: TabTitle=121-150
END_VISUALIZATION

// LMC_PacDrive/Application/TemplateFullProgrammingFramework/Visualization/Multicarrier/Vis_Positions_121_150
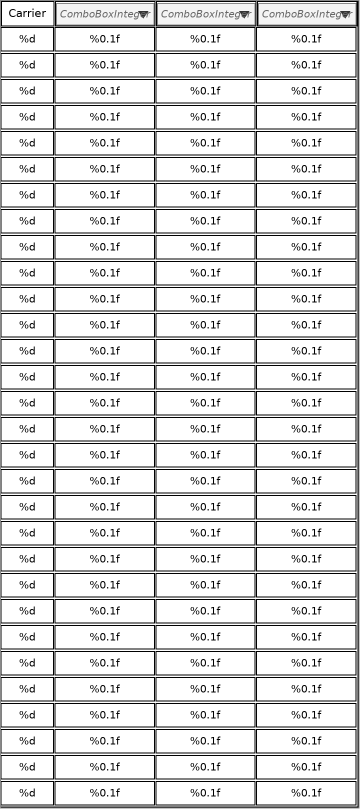
VISUALIZATION Vis_Positions_121_150  // 360x809
    Rectangle (0,0 358x807)
    Rectangle (55,1 100x25), "Position"
    Rectangle (257,1 100x25), "Gap Behind"
    Rectangle (1,1 53x25), "Carrier"
    Rectangle (156,1 100x25), "Gap In Front"
    Rectangle (55,1 100x25), "Position", invisible if: not SR_MultiCarriermodule.xInitSuccessful
    Rectangle (156,1 100x25), "Gap In Front", invisible if: not SR_MultiCarriermodule.xInitSuccessful
    Rectangle (257,1 100x25), "Gap Behind", invisible if: not SR_MultiCarriermodule.xInitSuccessful
    ComboBoxInteger (258,3 98x22), tooltip "RefTrackPosition RefPosition Gap to Carrier in front Distance to Carrier in front Gap to Carrier behind Distance to Carrier behind", variable: SR_MulticarrierModule.etVisPosColumn3, text list: 'TextList_VisPositions'
    ComboBoxInteger (157,3 98x22), tooltip "RefTrackPosition RefPosition Gap to Carrier in front Distance to Carrier in front Gap to Carrier behind Distance to Carrier behind", variable: SR_MulticarrierModule.etVisPosColumn2, text list: 'TextList_VisPositions'
    ComboBoxInteger (56,3 98x22), tooltip "RefTrackPosition RefPosition Gap to Carrier in front Distance to Carrier in front Gap to Carrier behind Distance to Carrier behind", variable: SR_MulticarrierModule.etVisPosColumn1, text list: 'TextList_VisPositions'
    Frame (0,27 358x26), invisible if: SR_MulticarrierModule.ifMulticarrier.ifFeedback.ifFeedbackConfiguration.udiNumberOfCarriers < 121 OR NOT SR_MultiCarriermodule.xInitSuccessful
        shows FR_CarDist(i_ifCarrierFeedback := SR_MultiCarrierModule.aifVisFeedback[121])
    Frame (0,53 358x26), invisible if: SR_MulticarrierModule.ifMulticarrier.ifFeedback.ifFeedbackConfiguration.udiNumberOfCarriers < 122 OR NOT SR_MultiCarriermodule.xInitSuccessful
        shows FR_CarDist(i_ifCarrierFeedback := SR_MultiCarrierModule.aifVisFeedback[122])
    Frame (0,79 358x26), invisible if: SR_MulticarrierModule.ifMulticarrier.ifFeedback.ifFeedbackConfiguration.udiNumberOfCarriers < 123 OR NOT SR_MultiCarriermodule.xInitSuccessful
        shows FR_CarDist(i_ifCarrierFeedback := SR_MultiCarrierModule.aifVisFeedback[123])
    Frame (0,105 358x26), invisible if: SR_MulticarrierModule.ifMulticarrier.ifFeedback.ifFeedbackConfiguration.udiNumberOfCarriers < 124 OR NOT SR_MultiCarriermodule.xInitSuccessful
        shows FR_CarDist(i_ifCarrierFeedback := SR_MultiCarrierModule.aifVisFeedback[124])
    Frame (0,131 358x26), invisible if: SR_MulticarrierModule.ifMulticarrier.ifFeedback.ifFeedbackConfiguration.udiNumberOfCarriers < 125 OR NOT SR_MultiCarriermodule.xInitSuccessful
        shows FR_CarDist(i_ifCarrierFeedback := SR_MultiCarrierModule.aifVisFeedback[125])
    Frame (0,157 358x26), invisible if: SR_MulticarrierModule.ifMulticarrier.ifFeedback.ifFeedbackConfiguration.udiNumberOfCarriers < 126 OR NOT SR_MultiCarriermodule.xInitSuccessful
        shows FR_CarDist(i_ifCarrierFeedback := SR_MultiCarrierModule.aifVisFeedback[126])
    Frame (0,183 358x26), invisible if: SR_MulticarrierModule.ifMulticarrier.ifFeedback.ifFeedbackConfiguration.udiNumberOfCarriers < 127 OR NOT SR_MultiCarriermodule.xInitSuccessful
        shows FR_CarDist(i_ifCarrierFeedback := SR_MultiCarrierModule.aifVisFeedback[127])
    Frame (0,209 358x26), invisible if: SR_MulticarrierModule.ifMulticarrier.ifFeedback.ifFeedbackConfiguration.udiNumberOfCarriers < 128 OR NOT SR_MultiCarriermodule.xInitSuccessful
        shows FR_CarDist(i_ifCarrierFeedback := SR_MultiCarrierModule.aifVisFeedback[128])
    Frame (0,235 358x26), invisible if: SR_MulticarrierModule.ifMulticarrier.ifFeedback.ifFeedbackConfiguration.udiNumberOfCarriers < 129 OR NOT SR_MultiCarriermodule.xInitSuccessful
        shows FR_CarDist(i_ifCarrierFeedback := SR_MultiCarrierModule.aifVisFeedback[129])
    Frame (0,261 358x26), invisible if: SR_MulticarrierModule.ifMulticarrier.ifFeedback.ifFeedbackConfiguration.udiNumberOfCarriers < 130 OR NOT SR_MultiCarriermodule.xInitSuccessful
        shows FR_CarDist(i_ifCarrierFeedback := SR_MultiCarrierModule.aifVisFeedback[130])
    Frame (0,287 358x26), invisible if: SR_MulticarrierModule.ifMulticarrier.ifFeedback.ifFeedbackConfiguration.udiNumberOfCarriers < 131 OR NOT SR_MultiCarriermodule.xInitSuccessful
        shows FR_CarDist(i_ifCarrierFeedback := SR_MultiCarrierModule.aifVisFeedback[131])
    Frame (0,313 358x26), invisible if: SR_MulticarrierModule.ifMulticarrier.ifFeedback.ifFeedbackConfiguration.udiNumberOfCarriers < 132 OR NOT SR_MultiCarriermodule.xInitSuccessful
        shows FR_CarDist(i_ifCarrierFeedback := SR_MultiCarrierModule.aifVisFeedback[132])
    Frame (0,339 358x26), invisible if: SR_MulticarrierModule.ifMulticarrier.ifFeedback.ifFeedbackConfiguration.udiNumberOfCarriers < 133 OR NOT SR_MultiCarriermodule.xInitSuccessful
        shows FR_CarDist(i_ifCarrierFeedback := SR_MultiCarrierModule.aifVisFeedback[133])
    Frame (0,365 358x26), invisible if: SR_MulticarrierModule.ifMulticarrier.ifFeedback.ifFeedbackConfiguration.udiNumberOfCarriers < 134 OR NOT SR_MultiCarriermodule.xInitSuccessful
        shows FR_CarDist(i_ifCarrierFeedback := SR_MultiCarrierModule.aifVisFeedback[134])
    Frame (0,391 358x26), invisible if: SR_MulticarrierModule.ifMulticarrier.ifFeedback.ifFeedbackConfiguration.udiNumberOfCarriers < 135 OR NOT SR_MultiCarriermodule.xInitSuccessful
        shows FR_CarDist(i_ifCarrierFeedback := SR_MultiCarrierModule.aifVisFeedback[135])
    Frame (0,417 358x26), invisible if: SR_MulticarrierModule.ifMulticarrier.ifFeedback.ifFeedbackConfiguration.udiNumberOfCarriers < 136 OR NOT SR_MultiCarriermodule.xInitSuccessful
        shows FR_CarDist(i_ifCarrierFeedback := SR_MultiCarrierModule.aifVisFeedback[136])
    Frame (0,443 358x26), invisible if: SR_MulticarrierModule.ifMulticarrier.ifFeedback.ifFeedbackConfiguration.udiNumberOfCarriers < 137 OR NOT SR_MultiCarriermodule.xInitSuccessful
        shows FR_CarDist(i_ifCarrierFeedback := SR_MultiCarrierModule.aifVisFeedback[137])
    Frame (0,469 358x26), invisible if: SR_MulticarrierModule.ifMulticarrier.ifFeedback.ifFeedbackConfiguration.udiNumberOfCarriers < 138 OR NOT SR_MultiCarriermodule.xInitSuccessful
        shows FR_CarDist(i_ifCarrierFeedback := SR_MultiCarrierModule.aifVisFeedback[138])
    Frame (0,495 358x26), invisible if: SR_MulticarrierModule.ifMulticarrier.ifFeedback.ifFeedbackConfiguration.udiNumberOfCarriers < 139 OR NOT SR_MultiCarriermodule.xInitSuccessful
        shows FR_CarDist(i_ifCarrierFeedback := SR_MultiCarrierModule.aifVisFeedback[139])
    Frame (0,521 358x26), invisible if: SR_MulticarrierModule.ifMulticarrier.ifFeedback.ifFeedbackConfiguration.udiNumberOfCarriers < 140 OR NOT SR_MultiCarriermodule.xInitSuccessful
        shows FR_CarDist(i_ifCarrierFeedback := SR_MultiCarrierModule.aifVisFeedback[140])
    Frame (0,547 358x26), invisible if: SR_MulticarrierModule.ifMulticarrier.ifFeedback.ifFeedbackConfiguration.udiNumberOfCarriers < 141 OR NOT SR_MultiCarriermodule.xInitSuccessful
        shows FR_CarDist(i_ifCarrierFeedback := SR_MultiCarrierModule.aifVisFeedback[141])
    Frame (0,573 358x26), invisible if: SR_MulticarrierModule.ifMulticarrier.ifFeedback.ifFeedbackConfiguration.udiNumberOfCarriers < 142 OR NOT SR_MultiCarriermodule.xInitSuccessful
        shows FR_CarDist(i_ifCarrierFeedback := SR_MultiCarrierModule.aifVisFeedback[142])
    Frame (0,599 358x26), invisible if: SR_MulticarrierModule.ifMulticarrier.ifFeedback.ifFeedbackConfiguration.udiNumberOfCarriers < 143 OR NOT SR_MultiCarriermodule.xInitSuccessful
        shows FR_CarDist(i_ifCarrierFeedback := SR_MultiCarrierModule.aifVisFeedback[143])
    Frame (0,625 358x26), invisible if: SR_MulticarrierModule.ifMulticarrier.ifFeedback.ifFeedbackConfiguration.udiNumberOfCarriers < 144 OR NOT SR_MultiCarriermodule.xInitSuccessful
        shows FR_CarDist(i_ifCarrierFeedback := SR_MultiCarrierModule.aifVisFeedback[144])
    Frame (0,651 358x26), invisible if: SR_MulticarrierModule.ifMulticarrier.ifFeedback.ifFeedbackConfiguration.udiNumberOfCarriers < 145 OR NOT SR_MultiCarriermodule.xInitSuccessful
        shows FR_CarDist(i_ifCarrierFeedback := SR_MultiCarrierModule.aifVisFeedback[145])
    Frame (0,677 358x26), invisible if: SR_MulticarrierModule.ifMulticarrier.ifFeedback.ifFeedbackConfiguration.udiNumberOfCarriers < 146 OR NOT SR_MultiCarriermodule.xInitSuccessful
        shows FR_CarDist(i_ifCarrierFeedback := SR_MultiCarrierModule.aifVisFeedback[146])
    Frame (0,703 358x26), invisible if: SR_MulticarrierModule.ifMulticarrier.ifFeedback.ifFeedbackConfiguration.udiNumberOfCarriers < 147 OR NOT SR_MultiCarriermodule.xInitSuccessful
        shows FR_CarDist(i_ifCarrierFeedback := SR_MultiCarrierModule.aifVisFeedback[147])
    Frame (0,729 358x26), invisible if: SR_MulticarrierModule.ifMulticarrier.ifFeedback.ifFeedbackConfiguration.udiNumberOfCarriers < 148 OR NOT SR_MultiCarriermodule.xInitSuccessful
        shows FR_CarDist(i_ifCarrierFeedback := SR_MultiCarrierModule.aifVisFeedback[148])
    Frame (0,755 358x26), invisible if: SR_MulticarrierModule.ifMulticarrier.ifFeedback.ifFeedbackConfiguration.udiNumberOfCarriers < 149 OR NOT SR_MultiCarriermodule.xInitSuccessful
        shows FR_CarDist(i_ifCarrierFeedback := SR_MultiCarrierModule.aifVisFeedback[149])
    Frame (0,781 358x26), invisible if: SR_MulticarrierModule.ifMulticarrier.ifFeedback.ifFeedbackConfiguration.udiNumberOfCarriers < 150 OR NOT SR_MultiCarriermodule.xInitSuccessful
        shows FR_CarDist(i_ifCarrierFeedback := SR_MultiCarrierModule.aifVisFeedback[150])
END_VISUALIZATION

// LMC_PacDrive/Application/TemplateFullProgrammingFramework/Visualization/Multicarrier/Vis_Positions_1_30
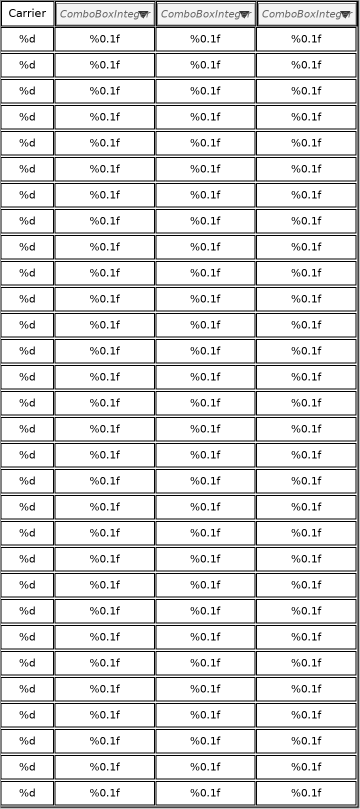
VISUALIZATION Vis_Positions_1_30  // 360x809
    Rectangle (0,0 358x807)
    Rectangle (1,1 53x25), "Carrier", invisible if: not SR_MultiCarriermodule.xInitSuccessful
    Frame (0,53 358x26), invisible if: SR_MulticarrierModule.ifMulticarrier.ifFeedback.ifFeedbackConfiguration.udiNumberOfCarriers < 2 OR NOT SR_MultiCarriermodule.xInitSuccessful
        shows FR_CarDist(i_ifCarrierFeedback := SR_MultiCarrierModule.aifVisFeedback[2])
    Frame (0,79 358x26), invisible if: SR_MulticarrierModule.ifMulticarrier.ifFeedback.ifFeedbackConfiguration.udiNumberOfCarriers < 3 OR NOT SR_MultiCarriermodule.xInitSuccessful
        shows FR_CarDist(i_ifCarrierFeedback := SR_MultiCarrierModule.aifVisFeedback[3])
    Frame (0,521 358x26), invisible if: SR_MulticarrierModule.ifMulticarrier.ifFeedback.ifFeedbackConfiguration.udiNumberOfCarriers < 20 OR NOT SR_MultiCarriermodule.xInitSuccessful
        shows FR_CarDist(i_ifCarrierFeedback := SR_MultiCarrierModule.aifVisFeedback[20])
    Frame (0,105 358x26), invisible if: SR_MulticarrierModule.ifMulticarrier.ifFeedback.ifFeedbackConfiguration.udiNumberOfCarriers < 4 OR NOT SR_MultiCarriermodule.xInitSuccessful
        shows FR_CarDist(i_ifCarrierFeedback := SR_MultiCarrierModule.aifVisFeedback[4])
    Frame (0,131 358x26), invisible if: SR_MulticarrierModule.ifMulticarrier.ifFeedback.ifFeedbackConfiguration.udiNumberOfCarriers < 5 OR NOT SR_MultiCarriermodule.xInitSuccessful
        shows FR_CarDist(i_ifCarrierFeedback := SR_MultiCarrierModule.aifVisFeedback[5])
    Frame (0,157 358x26), invisible if: SR_MulticarrierModule.ifMulticarrier.ifFeedback.ifFeedbackConfiguration.udiNumberOfCarriers < 6 OR NOT SR_MultiCarriermodule.xInitSuccessful
        shows FR_CarDist(i_ifCarrierFeedback := SR_MultiCarrierModule.aifVisFeedback[6])
    Frame (0,183 358x26), invisible if: SR_MulticarrierModule.ifMulticarrier.ifFeedback.ifFeedbackConfiguration.udiNumberOfCarriers < 7 OR NOT SR_MultiCarriermodule.xInitSuccessful
        shows FR_CarDist(i_ifCarrierFeedback := SR_MultiCarrierModule.aifVisFeedback[7])
    Frame (0,209 358x26), invisible if: SR_MulticarrierModule.ifMulticarrier.ifFeedback.ifFeedbackConfiguration.udiNumberOfCarriers < 8 OR NOT SR_MultiCarriermodule.xInitSuccessful
        shows FR_CarDist(i_ifCarrierFeedback := SR_MultiCarrierModule.aifVisFeedback[8])
    Frame (0,235 358x26), invisible if: SR_MulticarrierModule.ifMulticarrier.ifFeedback.ifFeedbackConfiguration.udiNumberOfCarriers < 9 OR NOT SR_MultiCarriermodule.xInitSuccessful
        shows FR_CarDist(i_ifCarrierFeedback := SR_MultiCarrierModule.aifVisFeedback[9])
    Frame (0,261 358x26), invisible if: SR_MulticarrierModule.ifMulticarrier.ifFeedback.ifFeedbackConfiguration.udiNumberOfCarriers < 10 OR NOT SR_MultiCarriermodule.xInitSuccessful
        shows FR_CarDist(i_ifCarrierFeedback := SR_MultiCarrierModule.aifVisFeedback[10])
    Frame (0,287 358x26), invisible if: SR_MulticarrierModule.ifMulticarrier.ifFeedback.ifFeedbackConfiguration.udiNumberOfCarriers < 11 OR NOT SR_MultiCarriermodule.xInitSuccessful
        shows FR_CarDist(i_ifCarrierFeedback := SR_MultiCarrierModule.aifVisFeedback[11])
    Frame (0,313 358x26), invisible if: SR_MulticarrierModule.ifMulticarrier.ifFeedback.ifFeedbackConfiguration.udiNumberOfCarriers < 12 OR NOT SR_MultiCarriermodule.xInitSuccessful
        shows FR_CarDist(i_ifCarrierFeedback := SR_MultiCarrierModule.aifVisFeedback[12])
    Frame (0,339 358x26), invisible if: SR_MulticarrierModule.ifMulticarrier.ifFeedback.ifFeedbackConfiguration.udiNumberOfCarriers < 13 OR NOT SR_MultiCarriermodule.xInitSuccessful
        shows FR_CarDist(i_ifCarrierFeedback := SR_MultiCarrierModule.aifVisFeedback[13])
    Frame (0,365 358x26), invisible if: SR_MulticarrierModule.ifMulticarrier.ifFeedback.ifFeedbackConfiguration.udiNumberOfCarriers < 14 OR NOT SR_MultiCarriermodule.xInitSuccessful
        shows FR_CarDist(i_ifCarrierFeedback := SR_MultiCarrierModule.aifVisFeedback[14])
    Frame (0,391 358x26), invisible if: SR_MulticarrierModule.ifMulticarrier.ifFeedback.ifFeedbackConfiguration.udiNumberOfCarriers < 15 OR NOT SR_MultiCarriermodule.xInitSuccessful
        shows FR_CarDist(i_ifCarrierFeedback := SR_MultiCarrierModule.aifVisFeedback[15])
    Frame (0,417 358x26), invisible if: SR_MulticarrierModule.ifMulticarrier.ifFeedback.ifFeedbackConfiguration.udiNumberOfCarriers < 16 OR NOT SR_MultiCarriermodule.xInitSuccessful
        shows FR_CarDist(i_ifCarrierFeedback := SR_MultiCarrierModule.aifVisFeedback[16])
    Frame (0,443 358x26), invisible if: SR_MulticarrierModule.ifMulticarrier.ifFeedback.ifFeedbackConfiguration.udiNumberOfCarriers < 17 OR NOT SR_MultiCarriermodule.xInitSuccessful
        shows FR_CarDist(i_ifCarrierFeedback := SR_MultiCarrierModule.aifVisFeedback[17])
    Frame (0,469 358x26), invisible if: SR_MulticarrierModule.ifMulticarrier.ifFeedback.ifFeedbackConfiguration.udiNumberOfCarriers < 18 OR NOT SR_MultiCarriermodule.xInitSuccessful
        shows FR_CarDist(i_ifCarrierFeedback := SR_MultiCarrierModule.aifVisFeedback[18])
    Frame (0,495 358x26), invisible if: SR_MulticarrierModule.ifMulticarrier.ifFeedback.ifFeedbackConfiguration.udiNumberOfCarriers < 19 OR NOT SR_MultiCarriermodule.xInitSuccessful
        shows FR_CarDist(i_ifCarrierFeedback := SR_MultiCarrierModule.aifVisFeedback[19])
    Frame (0,27 358x26), invisible if: SR_MulticarrierModule.ifMulticarrier.ifFeedback.ifFeedbackConfiguration.udiNumberOfCarriers < 1 OR NOT SR_MultiCarriermodule.xInitSuccessful
        shows FR_CarDist(i_ifCarrierFeedback := SR_MultiCarrierModule.aifVisFeedback[1])
    Rectangle (55,1 100x25), "Position", invisible if: not SR_MultiCarriermodule.xInitSuccessful
    Rectangle (156,1 100x25), "Gap In Front", invisible if: not SR_MultiCarriermodule.xInitSuccessful
    Rectangle (257,1 100x25), "Gap Behind", invisible if: not SR_MultiCarriermodule.xInitSuccessful
    ComboBoxInteger (258,3 98x22), tooltip "RefTrackPosition RefPosition Gap to Carrier in front Distance to Carrier in front Gap to Carrier behind Distance to Carrier behind", variable: SR_MulticarrierModule.etVisPosColumn3, text list: 'TextList_VisPositions'
    ComboBoxInteger (157,3 98x22), tooltip "RefTrackPosition RefPosition Gap to Carrier in front Distance to Carrier in front Gap to Carrier behind Distance to Carrier behind", variable: SR_MulticarrierModule.etVisPosColumn2, text list: 'TextList_VisPositions'
    ComboBoxInteger (56,3 98x22), tooltip "RefTrackPosition RefPosition Gap to Carrier in front Distance to Carrier in front Gap to Carrier behind Distance to Carrier behind", variable: SR_MulticarrierModule.etVisPosColumn1, text list: 'TextList_VisPositions'
    Frame (0,781 358x26), invisible if: SR_MulticarrierModule.ifMulticarrier.ifFeedback.ifFeedbackConfiguration.udiNumberOfCarriers < 30 OR NOT SR_MultiCarriermodule.xInitSuccessful
        shows FR_CarDist(i_ifCarrierFeedback := SR_MultiCarrierModule.aifVisFeedback[30])
    Frame (0,547 358x26), invisible if: SR_MulticarrierModule.ifMulticarrier.ifFeedback.ifFeedbackConfiguration.udiNumberOfCarriers < 21 OR NOT SR_MultiCarriermodule.xInitSuccessful
        shows FR_CarDist(i_ifCarrierFeedback := SR_MultiCarrierModule.aifVisFeedback[21])
    Frame (0,573 358x26), invisible if: SR_MulticarrierModule.ifMulticarrier.ifFeedback.ifFeedbackConfiguration.udiNumberOfCarriers < 22 OR NOT SR_MultiCarriermodule.xInitSuccessful
        shows FR_CarDist(i_ifCarrierFeedback := SR_MultiCarrierModule.aifVisFeedback[22])
    Frame (0,599 358x26), invisible if: SR_MulticarrierModule.ifMulticarrier.ifFeedback.ifFeedbackConfiguration.udiNumberOfCarriers < 23 OR NOT SR_MultiCarriermodule.xInitSuccessful
        shows FR_CarDist(i_ifCarrierFeedback := SR_MultiCarrierModule.aifVisFeedback[23])
    Frame (0,625 358x26), invisible if: SR_MulticarrierModule.ifMulticarrier.ifFeedback.ifFeedbackConfiguration.udiNumberOfCarriers < 24 OR NOT SR_MultiCarriermodule.xInitSuccessful
        shows FR_CarDist(i_ifCarrierFeedback := SR_MultiCarrierModule.aifVisFeedback[24])
    Frame (0,651 358x26), invisible if: SR_MulticarrierModule.ifMulticarrier.ifFeedback.ifFeedbackConfiguration.udiNumberOfCarriers < 25 OR NOT SR_MultiCarriermodule.xInitSuccessful
        shows FR_CarDist(i_ifCarrierFeedback := SR_MultiCarrierModule.aifVisFeedback[25])
    Frame (0,677 358x26), invisible if: SR_MulticarrierModule.ifMulticarrier.ifFeedback.ifFeedbackConfiguration.udiNumberOfCarriers < 26 OR NOT SR_MultiCarriermodule.xInitSuccessful
        shows FR_CarDist(i_ifCarrierFeedback := SR_MultiCarrierModule.aifVisFeedback[26])
    Frame (0,703 358x26), invisible if: SR_MulticarrierModule.ifMulticarrier.ifFeedback.ifFeedbackConfiguration.udiNumberOfCarriers < 27 OR NOT SR_MultiCarriermodule.xInitSuccessful
        shows FR_CarDist(i_ifCarrierFeedback := SR_MultiCarrierModule.aifVisFeedback[27])
    Frame (0,729 358x26), invisible if: SR_MulticarrierModule.ifMulticarrier.ifFeedback.ifFeedbackConfiguration.udiNumberOfCarriers < 28 OR NOT SR_MultiCarriermodule.xInitSuccessful
        shows FR_CarDist(i_ifCarrierFeedback := SR_MultiCarrierModule.aifVisFeedback[28])
    Frame (0,755 358x26), invisible if: SR_MulticarrierModule.ifMulticarrier.ifFeedback.ifFeedbackConfiguration.udiNumberOfCarriers < 29 OR NOT SR_MultiCarriermodule.xInitSuccessful
        shows FR_CarDist(i_ifCarrierFeedback := SR_MultiCarrierModule.aifVisFeedback[29])
END_VISUALIZATION

